# B&R Automation Studio project IP001
Automation Studio 4.7.3.93 SP

## Configuration Config1

CPU X20CP1301, AutomationRuntime C4.72, Build 4.1.2, Vc V4.72.0

### Hardware
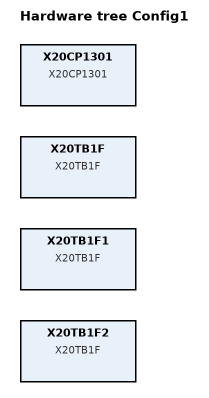
```
X20CP1301 : X20CP1301 v1.6.1.0  [X1 -> X1.SL; X2 -> X2.SL; X3 -> X3.SL]
  Module X1 (Type=X1, Virtual=true, Version=1.6.1.0)
    Connection (Connector=SS1, TargetModule=X20TB1F, TargetConnector=SS)
    Connection (Connector=SL, TargetModule=X20CP1301, TargetConnector=X1)
  Module X2 (Type=X2, Virtual=true, Version=1.6.1.0)
    Connection (Connector=SS1, TargetModule=X20TB1F1, TargetConnector=SS)
    Connection (Connector=SL, TargetModule=X20CP1301, TargetConnector=X2)
  Module X3 (Type=X3, Virtual=true, Version=1.6.1.0)
    Connection (Connector=SS1, TargetModule=X20TB1F2, TargetConnector=SS)
    Connection (Connector=SL, TargetModule=X20CP1301, TargetConnector=X3)
  Connector IF2:
    ActivateDevice = 1
    Mode = Manual
    InternetAddress = 192.168.15.199
    SubnetMask = 255.255.255.0
  ConfigurationID = IP001_Config1
  EthernetDefaultGateway = 192.168.15.254
  ActivateOpcUa = 1
  OpcUaInformationModels_PV_Version = 1
X20TB1F : X20TB1F v1.0.0.0
X20TB1F1 : X20TB1F v1.0.0.0
X20TB1F2 : X20TB1F v1.0.0.0
```

## Configuration DCS13_1

### Task classes (Cpu.sw)
```
Cyclic#4 (cycle 100000 us, tolerance 100000 us):
  DCS13_1 <- DCS13_1.prg
Libraries: Lib489, standard, AsMbTCP, operator, astime, AsIecCon, LibIP001, AsBrStr, asstring, MTBasics, DRV_mbus, DataObj, sys_lib, brsystem, MTTypes, dvframe, runtime
```

### Hardware
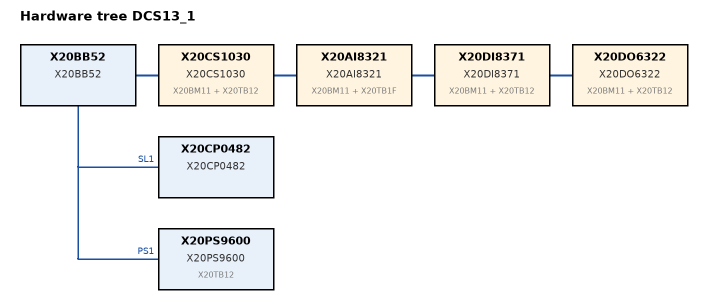
```
X20AI8321 : X20AI8321 v1.4.0.0  [SS1 -> X20TB1F.SS; SL -> X20BM11a.SL1]
X20BB52 : X20BB52 v1.1.0.0
X20BM11 : X20BM11 v1.0.0.1  [X2X1 -> X20BB52.IF6]
X20BM11a : X20BM11 v1.0.0.1  [X2X1 -> X20BM11.X2X2]
X20BM11b : X20BM11 v1.0.0.1  [X2X1 -> X20BM11a.X2X2]
X20BM11c : X20BM11 v1.0.0.1  [X2X1 -> X20BM11b.X2X2]
X20CP0482 : X20CP0482 v1.2.1.0  [SL -> X20BB52.SL1]
  Connector IF2:
    ActivateDevice = 1
    Mode = Manual
    InternetAddress = 192.168.50.15
    SubnetMask = 255.255.255.0
  ConfigurationID = IP001_DCS2_2
  TimerDeviceType = SWIOTIMER
  Cyclic1Duration = 10000
  Cyclic1Tolerance = 10000
  Cyclic2Duration = 20000
  Cyclic2Tolerance = 20000
  Cyclic3Duration = 50000
  Cyclic3Tolerance = 50000
  Cyclic4Duration = 100000
  Cyclic4Tolerance = 100000
  Cyclic5Duration = 200000
  Cyclic5Tolerance = 200000
  Cyclic6Duration = 500000
  Cyclic6Tolerance = 500000
  Cyclic7Duration = 1000000
  Cyclic7Tolerance = 1000000
  Cyclic8Duration = 10000
  Cyclic8Tolerance = 30000000
  ActivateOpcUa = 1
  OpcUa_AuthenticationSecurityPolicy_EnableNone = 1
  OpcUa_AuthenticationSecurityPolicy_EnableBasic128Rsa15 = 1
  OpcUaInformationModels_PV_Version = 1
X20CS1030 : X20CS1030 v1.7.0.0  [SS1 -> X20TB12a.SS; SL -> X20BM11.SL1]
X20DI8371 : X20DI8371 v1.0.2.0  [SS1 -> X20TB12b.SS; SL -> X20BM11b.SL1]
X20DO6322 : X20DO6322 v1.0.4.0  [SS1 -> X20TB12c.SS; SL -> X20BM11c.SL1]
X20PS9600 : X20PS9600 v1.0.2.0  [PS -> X20BB52.PS1; SS1 -> X20TB12.SS]
X20TB12 : X20TB12 v1.0.0.0
X20TB12a : X20TB12 v1.0.0.0
X20TB12b : X20TB12 v1.0.0.0
X20TB12c : X20TB12 v1.0.0.0
X20TB1F : X20TB1F v1.0.0.0
```

### IoMap.iom - X20CP0482/IoMap.iom
```iecst
VAR_CONFIG
	::DCS13_1:DI[1,1].In AT %IX."X20DI8371".DigitalInput01;
	::DCS13_1:DI[1,2].In AT %IX."X20DI8371".DigitalInput02;
	::DCS13_1:DI[1,3].In AT %IX."X20DI8371".DigitalInput03;
	::DCS13_1:DI[1,4].In AT %IX."X20DI8371".DigitalInput04;
	::DCS13_1:DO_[1,1].Out AT %QX."X20DO6322".DigitalOutput01;
	::DCS13_1:DO_[1,2].Out AT %QX."X20DO6322".DigitalOutput02;
	::DCS13_1:DO_[1,3].Out AT %QX."X20DO6322".DigitalOutput03;
	::DCS13_1:DO_[1,4].Out AT %QX."X20DO6322".DigitalOutput04;
	::DCS13_1:DO_[1,5].Out AT %QX."X20DO6322".DigitalOutput05;
	::DCS13_1:DO_[1,6].Out AT %QX."X20DO6322".DigitalOutput06;
	::DCS13_1:AI[1,1].RAW AT %IW."X20AI8321".AnalogInput01;
	::DCS13_1:AI[1,2].RAW AT %IW."X20AI8321".AnalogInput02;
	::DCS13_1:AI[1,3].RAW AT %IW."X20AI8321".AnalogInput03;
	::DCS13_1:AI[1,4].RAW AT %IW."X20AI8321".AnalogInput04;
	::DCS13_1:AI[1,5].RAW AT %IW."X20AI8321".AnalogInput05;
	::DCS13_1:AI[1,6].RAW AT %IW."X20AI8321".AnalogInput06;
	::DCS13_1:AI[1,7].RAW AT %IW."X20AI8321".AnalogInput07;
	::DCS13_1:AI[1,8].RAW AT %IW."X20AI8321".AnalogInput08;
	::DCS13_1:DI[1,5].In AT %IX."X20DI8371".DigitalInput05;
	::DCS13_1:DI[1,6].In AT %IX."X20DI8371".DigitalInput06;
	::DCS13_1:DI[1,7].In AT %IX."X20DI8371".DigitalInput07;
	::DCS13_1:DI[1,8].In AT %IX."X20DI8371".DigitalInput08;
END_VAR
```

## Configuration DCS15_1

CPU X20CP0482, AutomationRuntime C4.72, Build 4.1.2, Vc V4.72.0

### Task classes (Cpu.sw)
```
Cyclic#4 (cycle 100000 us, tolerance 100000 us):
  DCS15_1 <- DCS15_1.prg
Libraries: Lib489, standard, AsMbTCP, AsBrStr, asstring, operator, astime, AsIecCon, LibIP001, MTBasics, DRV_mbus, DataObj, sys_lib, brsystem, MTTypes, dvframe, runtime
```

### Hardware
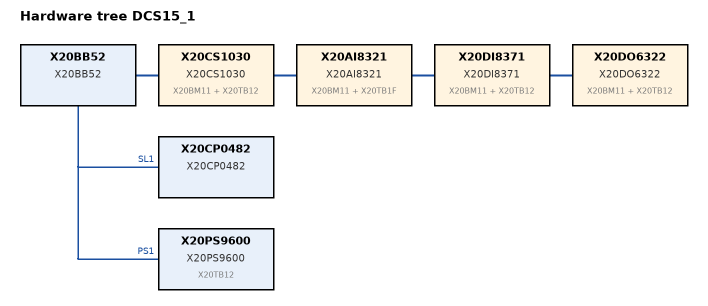
```
X20AI8321 : X20AI8321 v1.4.0.0  [SS1 -> X20TB1F.SS; SL -> X20BM11a.SL1]
X20BB52 : X20BB52 v1.1.0.0
X20BM11 : X20BM11 v1.0.0.1  [X2X1 -> X20BB52.IF6]
X20BM11a : X20BM11 v1.0.0.1  [X2X1 -> X20BM11.X2X2]
X20BM11b : X20BM11 v1.0.0.1  [X2X1 -> X20BM11a.X2X2]
X20BM11c : X20BM11 v1.0.0.1  [X2X1 -> X20BM11b.X2X2]
X20CP0482 : X20CP0482 v1.2.1.0  [SL -> X20BB52.SL1]
  Connector IF2:
    ActivateDevice = 1
    Mode = Manual
    InternetAddress = 192.168.50.16
    SubnetMask = 255.255.255.0
  ConfigurationID = IP001_DCS2_2
  TimerDeviceType = SWIOTIMER
  Cyclic1Duration = 10000
  Cyclic1Tolerance = 10000
  Cyclic2Duration = 20000
  Cyclic2Tolerance = 20000
  Cyclic3Duration = 50000
  Cyclic3Tolerance = 50000
  Cyclic4Duration = 100000
  Cyclic4Tolerance = 100000
  Cyclic5Duration = 200000
  Cyclic5Tolerance = 200000
  Cyclic6Duration = 500000
  Cyclic6Tolerance = 500000
  Cyclic7Duration = 1000000
  Cyclic7Tolerance = 1000000
  Cyclic8Duration = 10000
  Cyclic8Tolerance = 30000000
  ActivateOpcUa = 1
  OpcUa_AuthenticationSecurityPolicy_EnableNone = 1
  OpcUa_AuthenticationSecurityPolicy_EnableBasic128Rsa15 = 1
  OpcUaInformationModels_PV_Version = 1
X20CS1030 : X20CS1030 v1.7.0.0  [SS1 -> X20TB12a.SS; SL -> X20BM11.SL1]
X20DI8371 : X20DI8371 v1.0.2.0  [SS1 -> X20TB12b.SS; SL -> X20BM11b.SL1]
X20DO6322 : X20DO6322 v1.0.4.0  [SS1 -> X20TB12c.SS; SL -> X20BM11c.SL1]
X20PS9600 : X20PS9600 v1.0.2.0  [PS -> X20BB52.PS1; SS1 -> X20TB12.SS]
X20TB12 : X20TB12 v1.0.0.0
X20TB12a : X20TB12 v1.0.0.0
X20TB12b : X20TB12 v1.0.0.0
X20TB12c : X20TB12 v1.0.0.0
X20TB1F : X20TB1F v1.0.0.0
```

### IoMap.iom - X20CP0482/IoMap.iom
```iecst
VAR_CONFIG
	::DCS15_1:DI[1,1].In AT %IX."X20DI8371".DigitalInput01;
	::DCS15_1:DI[1,2].In AT %IX."X20DI8371".DigitalInput02;
	::DCS15_1:DI[1,3].In AT %IX."X20DI8371".DigitalInput03;
	::DCS15_1:DI[1,4].In AT %IX."X20DI8371".DigitalInput04;
	::DCS15_1:DO_[1,1].Out AT %QX."X20DO6322".DigitalOutput01;
	::DCS15_1:DO_[1,2].Out AT %QX."X20DO6322".DigitalOutput02;
	::DCS15_1:DO_[1,3].Out AT %QX."X20DO6322".DigitalOutput03;
	::DCS15_1:DO_[1,4].Out AT %QX."X20DO6322".DigitalOutput04;
	::DCS15_1:DO_[1,5].Out AT %QX."X20DO6322".DigitalOutput05;
	::DCS15_1:DO_[1,6].Out AT %QX."X20DO6322".DigitalOutput06;
	::DCS15_1:AI[1,1].RAW AT %IW."X20AI8321".AnalogInput01;
	::DCS15_1:AI[1,2].RAW AT %IW."X20AI8321".AnalogInput02;
	::DCS15_1:AI[1,3].RAW AT %IW."X20AI8321".AnalogInput03;
	::DCS15_1:AI[1,4].RAW AT %IW."X20AI8321".AnalogInput04;
	::DCS15_1:AI[1,5].RAW AT %IW."X20AI8321".AnalogInput05;
	::DCS15_1:AI[1,6].RAW AT %IW."X20AI8321".AnalogInput06;
	::DCS15_1:AI[1,7].RAW AT %IW."X20AI8321".AnalogInput07;
	::DCS15_1:AI[1,8].RAW AT %IW."X20AI8321".AnalogInput08;
	::DCS15_1:DI[1,5].In AT %IX."X20DI8371".DigitalInput05;
	::DCS15_1:DI[1,6].In AT %IX."X20DI8371".DigitalInput06;
	::DCS15_1:DI[1,7].In AT %IX."X20DI8371".DigitalInput07;
	::DCS15_1:DI[1,8].In AT %IX."X20DI8371".DigitalInput08;
END_VAR
```

## Configuration DCS18_1

### Hardware
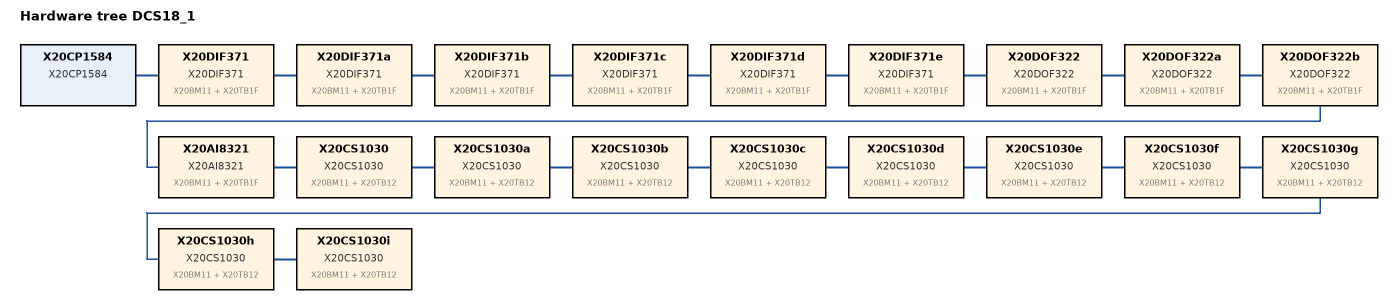
```
X20AI8321 : X20AI8321 v1.4.0.0  [SS1 -> X20TB1F.SS; SL -> X20BM11a.SL1]
X20BM11 : X20BM11 v1.0.0.1  [X2X1 -> X20BM11a.X2X2]
X20BM11a : X20BM11 v1.0.0.1  [X2X1 -> X20BM11l.X2X2]
X20BM11b : X20BM11 v1.0.0.1  [X2X1 -> X20CP1584.IF6]
X20BM11c : X20BM11 v1.0.0.1  [X2X1 -> X20BM11m.X2X2]
X20BM11d : X20BM11 v1.0.0.1  [X2X1 -> X20BM11g.X2X2]
X20BM11e : X20BM11 v1.0.0.1  [X2X1 -> X20BM11d.X2X2]
X20BM11f : X20BM11 v1.0.0.1  [X2X1 -> X20BM11c.X2X2]
X20BM11g : X20BM11 v1.0.0.1  [X2X1 -> X20BM11.X2X2]
X20BM11h : X20BM11 v1.0.0.1  [X2X1 -> X20BM11b.X2X2]
X20BM11i : X20BM11 v1.0.0.1  [X2X1 -> X20BM11h.X2X2]
X20BM11j : X20BM11 v1.0.0.1  [X2X1 -> X20BM11i.X2X2]
X20BM11k : X20BM11 v1.0.0.1  [X2X1 -> X20BM11j.X2X2]
X20BM11l : X20BM11 v1.0.0.1  [X2X1 -> X20BM11f.X2X2]
X20BM11m : X20BM11 v1.0.0.1  [X2X1 -> X20BM11k.X2X2]
X20BM11n : X20BM11 v1.0.0.1  [X2X1 -> X20BM11e.X2X2]
X20BM11o : X20BM11 v1.0.0.1  [X2X1 -> X20BM11n.X2X2]
X20BM11p : X20BM11 v1.0.0.1  [X2X1 -> X20BM11o.X2X2]
X20BM11q : X20BM11 v1.0.0.1  [X2X1 -> X20BM11p.X2X2]
X20BM11r : X20BM11 v1.0.0.1  [X2X1 -> X20BM11q.X2X2]
X20BM11s : X20BM11 v1.0.0.1  [X2X1 -> X20BM11r.X2X2]
X20CP1584 : X20CP1584 v1.8.0.0
  Connector IF2:
    ActivateDevice = 1
    Mode = Manual
    InternetAddress = 192.168.50.17
    SubnetMask = 255.255.255.0
  ConfigurationID = IP001_DCS2_2
  ActivateOpcUa = 1
  OpcUa_AuthenticationSecurityPolicy_EnableNone = 1
  OpcUa_AuthenticationSecurityPolicy_EnableBasic128Rsa15 = 1
  OpcUaInformationModels_PV_Version = 1
X20CS1030 : X20CS1030 v1.7.0.0  [SS1 -> X20TB12a.SS; SL -> X20BM11.SL1]
X20CS1030a : X20CS1030 v1.7.0.0  [SS1 -> X20TB12.SS; SL -> X20BM11g.SL1]
X20CS1030b : X20CS1030 v1.7.0.0  [SS1 -> X20TB12b.SS; SL -> X20BM11d.SL1]
X20CS1030c : X20CS1030 v1.7.0.0  [SS1 -> X20TB12c.SS; SL -> X20BM11e.SL1]
X20CS1030d : X20CS1030 v1.7.0.0  [SS1 -> X20TB12d.SS; SL -> X20BM11n.SL1]
X20CS1030e : X20CS1030 v1.7.0.0  [SS1 -> X20TB12e.SS; SL -> X20BM11o.SL1]
X20CS1030f : X20CS1030 v1.7.0.0  [SS1 -> X20TB12f.SS; SL -> X20BM11p.SL1]
X20CS1030g : X20CS1030 v1.7.0.0  [SS1 -> X20TB12g.SS; SL -> X20BM11q.SL1]
X20CS1030h : X20CS1030 v1.7.0.0  [SS1 -> X20TB12h.SS; SL -> X20BM11r.SL1]
X20CS1030i : X20CS1030 v1.7.0.0  [SS1 -> X20TB12i.SS; SL -> X20BM11s.SL1]
X20DIF371 : X20DIF371 v1.1.0.0  [SS1 -> X20TB1F1.SS; SL -> X20BM11b.SL1]
X20DIF371a : X20DIF371 v1.1.0.0  [SS1 -> X20TB1F2.SS; SL -> X20BM11h.SL1]
X20DIF371b : X20DIF371 v1.1.0.0  [SS1 -> X20TB1F3.SS; SL -> X20BM11i.SL1]
X20DIF371c : X20DIF371 v1.1.0.0  [SS1 -> X20TB1F4.SS; SL -> X20BM11j.SL1]
X20DIF371d : X20DIF371 v1.1.0.0  [SS1 -> X20TB1F5.SS; SL -> X20BM11k.SL1]
X20DIF371e : X20DIF371 v1.1.0.0  [SS1 -> X20TB1F9.SS; SL -> X20BM11m.SL1]
X20DOF322 : X20DOF322 v1.4.0.0  [SS1 -> X20TB1F6.SS; SL -> X20BM11c.SL1]
X20DOF322a : X20DOF322 v1.4.0.0  [SS1 -> X20TB1F7.SS; SL -> X20BM11f.SL1]
X20DOF322b : X20DOF322 v1.4.0.0  [SS1 -> X20TB1F8.SS; SL -> X20BM11l.SL1]
X20TB12 : X20TB12 v1.0.0.0
X20TB12a : X20TB12 v1.0.0.0
X20TB12b : X20TB12 v1.0.0.0
X20TB12c : X20TB12 v1.0.0.0
X20TB12d : X20TB12 v1.0.0.0
X20TB12e : X20TB12 v1.0.0.0
X20TB12f : X20TB12 v1.0.0.0
X20TB12g : X20TB12 v1.0.0.0
X20TB12h : X20TB12 v1.0.0.0
X20TB12i : X20TB12 v1.0.0.0
X20TB1F : X20TB1F v1.0.0.0
X20TB1F1 : X20TB1F v1.0.0.0
X20TB1F2 : X20TB1F v1.0.0.0
X20TB1F3 : X20TB1F v1.0.0.0
X20TB1F4 : X20TB1F v1.0.0.0
X20TB1F5 : X20TB1F v1.0.0.0
X20TB1F6 : X20TB1F v1.0.0.0
X20TB1F7 : X20TB1F v1.0.0.0
X20TB1F8 : X20TB1F v1.0.0.0
X20TB1F9 : X20TB1F v1.0.0.0
```

### IoMap.iom - X20CP1584/IoMap.iom
```iecst
VAR_CONFIG
	::DCS18_1:AI[1,1].RAW AT %IW."X20AI8321".AnalogInput01;
	::DCS18_1:AI[1,2].RAW AT %IW."X20AI8321".AnalogInput02;
	::DCS18_1:AI[1,3].RAW AT %IW."X20AI8321".AnalogInput03;
	::DCS18_1:AI[1,4].RAW AT %IW."X20AI8321".AnalogInput04;
	::DCS18_1:AI[1,5].RAW AT %IW."X20AI8321".AnalogInput05;
	::DCS18_1:AI[1,6].RAW AT %IW."X20AI8321".AnalogInput06;
	::DCS18_1:AI[1,7].RAW AT %IW."X20AI8321".AnalogInput07;
	::DCS18_1:AI[1,8].RAW AT %IW."X20AI8321".AnalogInput08;
	::DCS18_1:DI[1,1].In AT %IX."X20DIF371".DigitalInput01;
	::DCS18_1:DI[1,2].In AT %IX."X20DIF371".DigitalInput02;
	::DCS18_1:DI[1,3].In AT %IX."X20DIF371".DigitalInput03;
	::DCS18_1:DI[1,4].In AT %IX."X20DIF371".DigitalInput04;
	::DCS18_1:DI[1,5].In AT %IX."X20DIF371".DigitalInput05;
	::DCS18_1:DI[1,6].In AT %IX."X20DIF371".DigitalInput06;
	::DCS18_1:DI[1,7].In AT %IX."X20DIF371".DigitalInput07;
	::DCS18_1:DI[1,8].In AT %IX."X20DIF371".DigitalInput08;
	::DCS18_1:DI[1,9].In AT %IX."X20DIF371".DigitalInput09;
	::DCS18_1:DI[1,10].In AT %IX."X20DIF371".DigitalInput10;
	::DCS18_1:DI[1,11].In AT %IX."X20DIF371".DigitalInput11;
	::DCS18_1:DI[1,12].In AT %IX."X20DIF371".DigitalInput12;
	::DCS18_1:DI[1,13].In AT %IX."X20DIF371".DigitalInput13;
	::DCS18_1:DI[1,14].In AT %IX."X20DIF371".DigitalInput14;
	::DCS18_1:DI[1,15].In AT %IX."X20DIF371".DigitalInput15;
	::DCS18_1:DI[1,16].In AT %IX."X20DIF371".DigitalInput16;
	::DCS18_1:DO_[1,1].Out AT %QX."X20DOF322".DigitalOutput01;
	::DCS18_1:DO_[1,2].Out AT %QX."X20DOF322".DigitalOutput02;
	::DCS18_1:DO_[1,3].Out AT %QX."X20DOF322".DigitalOutput03;
	::DCS18_1:DO_[1,4].Out AT %QX."X20DOF322".DigitalOutput04;
	::DCS18_1:DO_[1,5].Out AT %QX."X20DOF322".DigitalOutput05;
	::DCS18_1:DO_[1,6].Out AT %QX."X20DOF322".DigitalOutput06;
	::DCS18_1:DO_[1,7].Out AT %QX."X20DOF322".DigitalOutput07;
	::DCS18_1:DO_[1,8].Out AT %QX."X20DOF322".DigitalOutput08;
	::DCS18_1:DO_[1,9].Out AT %QX."X20DOF322".DigitalOutput09;
	::DCS18_1:DO_[1,10].Out AT %QX."X20DOF322".DigitalOutput10;
	::DCS18_1:DO_[1,11].Out AT %QX."X20DOF322".DigitalOutput11;
	::DCS18_1:DO_[1,12].Out AT %QX."X20DOF322".DigitalOutput12;
	::DCS18_1:DO_[1,13].Out AT %QX."X20DOF322".DigitalOutput13;
	::DCS18_1:DO_[1,14].Out AT %QX."X20DOF322".DigitalOutput14;
	::DCS18_1:DO_[1,15].Out AT %QX."X20DOF322".DigitalOutput15;
	::DCS18_1:DO_[1,16].Out AT %QX."X20DOF322".DigitalOutput16;
	::DCS18_1:DO_[2,1].Out AT %QX."X20DOF322a".DigitalOutput01;
	::DCS18_1:DO_[2,2].Out AT %QX."X20DOF322a".DigitalOutput02;
	::DCS18_1:DO_[2,3].Out AT %QX."X20DOF322a".DigitalOutput03;
	::DCS18_1:DO_[2,4].Out  AT %QX."X20DOF322a".DigitalOutput04;
	::DCS18_1:DO_[2,5].Out  AT %QX."X20DOF322a".DigitalOutput05;
	::DCS18_1:DO_[2,6].Out  AT %QX."X20DOF322a".DigitalOutput06;
	::DCS18_1:DO_[2,7].Out  AT %QX."X20DOF322a".DigitalOutput07;
	::DCS18_1:DO_[2,8].Out  AT %QX."X20DOF322a".DigitalOutput08;
	::DCS18_1:DO_[2,9].Out  AT %QX."X20DOF322a".DigitalOutput09;
	::DCS18_1:DO_[2,10].Out  AT %QX."X20DOF322a".DigitalOutput10;
	::DCS18_1:DO_[2,11].Out  AT %QX."X20DOF322a".DigitalOutput11;
	::DCS18_1:DO_[2,12].Out  AT %QX."X20DOF322a".DigitalOutput12;
	::DCS18_1:DO_[2,13].Out  AT %QX."X20DOF322a".DigitalOutput13;
	::DCS18_1:DO_[2,14].Out  AT %QX."X20DOF322a".DigitalOutput14;
	::DCS18_1:DO_[2,15].Out  AT %QX."X20DOF322a".DigitalOutput15;
	::DCS18_1:DO_[2,16].Out  AT %QX."X20DOF322a".DigitalOutput16;
	::DCS18_1:DO_[3,1].Out AT %QX."X20DOF322b".DigitalOutput01;
	::DCS18_1:DO_[3,2].Out  AT %QX."X20DOF322b".DigitalOutput02;
	::DCS18_1:DO_[3,3].Out  AT %QX."X20DOF322b".DigitalOutput03;
	::DCS18_1:DO_[3,4].Out  AT %QX."X20DOF322b".DigitalOutput04;
	::DCS18_1:DO_[3,5].Out  AT %QX."X20DOF322b".DigitalOutput05;
	::DCS18_1:DO_[3,6].Out  AT %QX."X20DOF322b".DigitalOutput06;
	::DCS18_1:DO_[3,7].Out  AT %QX."X20DOF322b".DigitalOutput07;
	::DCS18_1:DO_[3,8].Out  AT %QX."X20DOF322b".DigitalOutput08;
	::DCS18_1:DO_[3,9].Out  AT %QX."X20DOF322b".DigitalOutput09;
	::DCS18_1:DO_[3,10].Out  AT %QX."X20DOF322b".DigitalOutput10;
	::DCS18_1:DO_[3,11].Out  AT %QX."X20DOF322b".DigitalOutput11;
	::DCS18_1:DO_[3,12].Out  AT %QX."X20DOF322b".DigitalOutput12;
	::DCS18_1:DO_[3,13].Out  AT %QX."X20DOF322b".DigitalOutput13;
	::DCS18_1:DO_[3,14].Out  AT %QX."X20DOF322b".DigitalOutput14;
	::DCS18_1:DO_[3,15].Out  AT %QX."X20DOF322b".DigitalOutput15;
	::DCS18_1:DO_[3,16].Out  AT %QX."X20DOF322b".DigitalOutput16;
END_VAR
```

## Configuration DCS2_2

CPU X20CP0482, AutomationRuntime B4.92, Build 4.1.2, Vc V4.72.5

### Task classes (Cpu.sw)
```
Cyclic#4 (cycle 100000 us, tolerance 100000 us):
  DCS2_2 <- DCS2_2.prg
Libraries: Lib489, standard, AsMbTCP, AsBrStr, asstring, MTBasics, DRV_mbus, DataObj, sys_lib, brsystem, MTTypes, dvframe, runtime, LibIP001
```

### Hardware
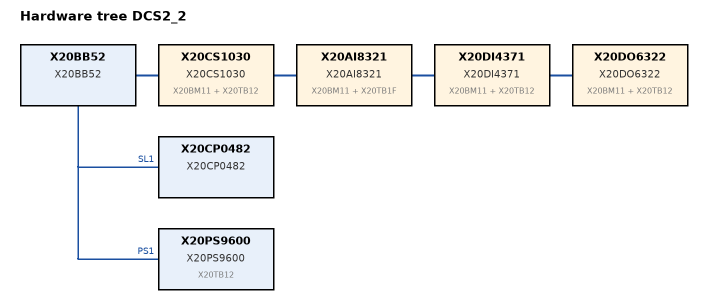
```
X20AI8321 : X20AI8321 v1.5.0.0  [SS1 -> X20TB1F.SS; SL -> X20BM11a.SL1]
X20BB52 : X20BB52 v1.2.0.0
X20BM11 : X20BM11 v1.1.0.0  [X2X1 -> X20BB52.IF6]
X20BM11a : X20BM11 v1.1.0.0  [X2X1 -> X20BM11.X2X2]
X20BM11b : X20BM11 v1.1.0.0  [X2X1 -> X20BM11a.X2X2]
X20BM11c : X20BM11 v1.1.0.0  [X2X1 -> X20BM11b.X2X2]
X20CP0482 : X20CP0482 v1.5.0.0  [SL -> X20BB52.SL1]
  Connector IF2:
    ActivateDevice = 1
    Mode = Manual
    InternetAddress = 192.168.50.10
    SubnetMask = 255.255.255.0
  Connector IF3:
    DNAConfiguration = manual
  ConfigurationID = IP001_DCS2_2
  UserPartitionSize = 0
  Simulation = 1
  TimerDeviceType = SWIOTIMER
  Cyclic1Duration = 10000
  Cyclic1Tolerance = 10000
  Cyclic2Duration = 20000
  Cyclic2Tolerance = 20000
  Cyclic3Duration = 50000
  Cyclic3Tolerance = 50000
  Cyclic4Duration = 100000
  Cyclic4Tolerance = 100000
  Cyclic5Duration = 200000
  Cyclic5Tolerance = 200000
  Cyclic6Duration = 500000
  Cyclic6Tolerance = 500000
  Cyclic7Duration = 1000000
  Cyclic7Tolerance = 1000000
  Cyclic8Duration = 10000
  Cyclic8Tolerance = 30000000
  FileDevice1
  FileDeviceName1 = USER
  FileDevicePath1 = USER_PATH
  ActivateOpcUa = 1
  OpcUa_AuthenticationSecurityPolicy_EnableNone = 1
  OpcUa_AuthenticationSecurityPolicy_EnableBasic128Rsa15 = 1
  OpcUaInformationModels_PV_Version = 1
X20CS1030 : X20CS1030 v1.8.0.0  [SS1 -> X20TB12a.SS; SL -> X20BM11.SL1]
X20DI4371 : X20DI4371 v1.2.0.0  [SS1 -> X20TB12b.SS; SL -> X20BM11b.SL1]
X20DO6322 : X20DO6322 v1.2.0.0  [SS1 -> X20TB12c.SS; SL -> X20BM11c.SL1]
X20PS9600 : X20PS9600 v1.6.0.0  [PS -> X20BB52.PS1; SS1 -> X20TB12.SS]
X20TB12 : X20TB12 v1.0.0.0
X20TB12a : X20TB12 v1.0.0.0
X20TB12b : X20TB12 v1.0.0.0
X20TB12c : X20TB12 v1.0.0.0
X20TB1F : X20TB1F v1.0.0.0
```

### IoMap.iom - X20CP0482/IoMap.iom
```iecst
VAR_CONFIG
	::DCS2_2:AI[1,1].RAW AT %IW."X20AI8321".AnalogInput01;
	::DCS2_2:AI[1,2].RAW  AT %IW."X20AI8321".AnalogInput02;
	::DCS2_2:AI[1,3].RAW AT %IW."X20AI8321".AnalogInput03;
	::DCS2_2:AI[1,4].RAW AT %IW."X20AI8321".AnalogInput04;
	::DCS2_2:AI[1,5].RAW AT %IW."X20AI8321".AnalogInput05;
	::DCS2_2:AI[1,6].RAW AT %IW."X20AI8321".AnalogInput06;
	::DCS2_2:AI[1,7].RAW AT %IW."X20AI8321".AnalogInput07;
	::DCS2_2:AI[1,8].RAW AT %IW."X20AI8321".AnalogInput08;
	::DCS2_2:DI[1,1].In AT %IX."X20DI4371".DigitalInput01;
	::DCS2_2:DI[1,2].In AT %IX."X20DI4371".DigitalInput02;
	::DCS2_2:DI[1,3].In AT %IX."X20DI4371".DigitalInput03;
	::DCS2_2:DI[1,4].In AT %IX."X20DI4371".DigitalInput04;
	::DCS2_2:DO_[1,1].Out AT %QX."X20DO6322".DigitalOutput01;
	::DCS2_2:DO_[1,2].Out AT %QX."X20DO6322".DigitalOutput02;
	::DCS2_2:DO_[1,3].Out AT %QX."X20DO6322".DigitalOutput03;
	::DCS2_2:DO_[1,4].Out AT %QX."X20DO6322".DigitalOutput04;
	::DCS2_2:DO_[1,5].Out AT %QX."X20DO6322".DigitalOutput05;
	::DCS2_2:DO_[1,6].Out AT %QX."X20DO6322".DigitalOutput06;
END_VAR
```

## Configuration DCS31_1

CPU X20CP0482, AutomationRuntime C4.72, Build 4.1.2, Vc V4.72.0

### Task classes (Cpu.sw)
```
Cyclic#4 (cycle 100000 us, tolerance 100000 us):
  DCS31_1 <- DCS31_1.prg
Libraries: Lib489, standard, AsMbTCP, AsBrStr, asstring, operator, astime, AsIecCon, LibIP001, MTBasics, DRV_mbus, DataObj, sys_lib, brsystem, MTTypes, dvframe, runtime
```

### Hardware
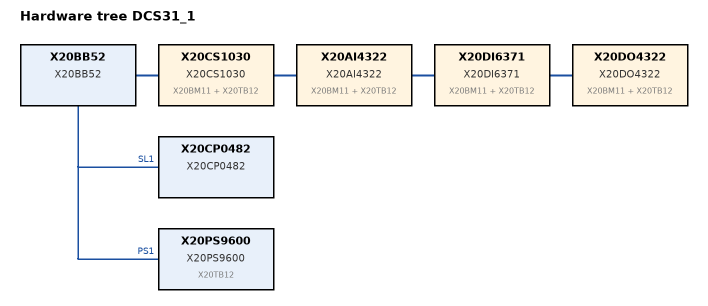
```
X20AI4322 : X20AI4322 v1.0.0.2  [SS1 -> X20TB12d.SS; SL -> X20BM11a.SL1]
X20BB52 : X20BB52 v1.1.0.0
X20BM11 : X20BM11 v1.0.0.1  [X2X1 -> X20BB52.IF6]
X20BM11a : X20BM11 v1.0.0.1  [X2X1 -> X20BM11.X2X2]
X20BM11b : X20BM11 v1.0.0.1  [X2X1 -> X20BM11a.X2X2]
X20BM11c : X20BM11 v1.0.0.1  [X2X1 -> X20BM11b.X2X2]
X20CP0482 : X20CP0482 v1.2.1.0  [SL -> X20BB52.SL1]
  Connector IF2:
    ActivateDevice = 1
    Mode = Manual
    InternetAddress = 192.168.50.18
    SubnetMask = 255.255.255.0
  ConfigurationID = IP001_DCS2_2
  TimerDeviceType = SWIOTIMER
  Cyclic1Duration = 10000
  Cyclic1Tolerance = 10000
  Cyclic2Duration = 20000
  Cyclic2Tolerance = 20000
  Cyclic3Duration = 50000
  Cyclic3Tolerance = 50000
  Cyclic4Duration = 100000
  Cyclic4Tolerance = 100000
  Cyclic5Duration = 200000
  Cyclic5Tolerance = 200000
  Cyclic6Duration = 500000
  Cyclic6Tolerance = 500000
  Cyclic7Duration = 1000000
  Cyclic7Tolerance = 1000000
  Cyclic8Duration = 10000
  Cyclic8Tolerance = 30000000
  ActivateOpcUa = 1
  OpcUa_AuthenticationSecurityPolicy_EnableNone = 1
  OpcUa_AuthenticationSecurityPolicy_EnableBasic128Rsa15 = 1
  OpcUaInformationModels_PV_Version = 1
X20CS1030 : X20CS1030 v1.7.0.0  [SS1 -> X20TB12a.SS; SL -> X20BM11.SL1]
X20DI6371 : X20DI6371 v1.0.2.0  [SS1 -> X20TB12b.SS; SL -> X20BM11b.SL1]
X20DO4322 : X20DO4322 v1.0.3.0  [SS1 -> X20TB12c.SS; SL -> X20BM11c.SL1]
X20PS9600 : X20PS9600 v1.0.2.0  [PS -> X20BB52.PS1; SS1 -> X20TB12.SS]
X20TB12 : X20TB12 v1.0.0.0
X20TB12a : X20TB12 v1.0.0.0
X20TB12b : X20TB12 v1.0.0.0
X20TB12c : X20TB12 v1.0.0.0
X20TB12d : X20TB12 v1.0.0.0
```

### IoMap.iom - X20CP0482/IoMap.iom
```iecst
VAR_CONFIG
	::DCS31_1:DI[1,1].In AT %IX."X20DI6371".DigitalInput01;
	::DCS31_1:DI[1,2].In AT %IX."X20DI6371".DigitalInput02;
	::DCS31_1:DI[1,3].In AT %IX."X20DI6371".DigitalInput03;
	::DCS31_1:DI[1,4].In AT %IX."X20DI6371".DigitalInput04;
	::DCS31_1:DO_[1,1].Out AT %QX."X20DO4322".DigitalOutput01;
	::DCS31_1:DO_[1,2].Out AT %QX."X20DO4322".DigitalOutput02;
	::DCS31_1:DO_[1,3].Out AT %QX."X20DO4322".DigitalOutput03;
	::DCS31_1:DO_[1,4].Out AT %QX."X20DO4322".DigitalOutput04;
	::DCS31_1:AI[1,1].RAW AT %IW."X20AI4322".AnalogInput01;
	::DCS31_1:AI[1,2].RAW AT %IW."X20AI4322".AnalogInput02;
	::DCS31_1:AI[1,3].RAW AT %IW."X20AI4322".AnalogInput03;
	::DCS31_1:AI[1,4].RAW AT %IW."X20AI4322".AnalogInput04;
	::DCS31_1:DI[1,5].In AT %IX."X20DI6371".DigitalInput05;
	::DCS31_1:DI[1,6].In AT %IX."X20DI6371".DigitalInput06;
END_VAR
```

## Configuration DCS31_2

### Hardware
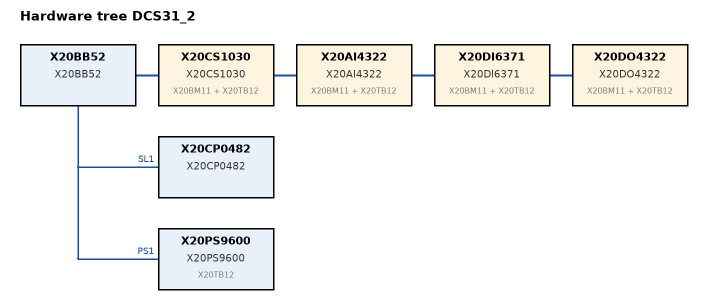
```
X20AI4322 : X20AI4322 v1.0.0.2  [SS1 -> X20TB12d.SS; SL -> X20BM11a.SL1]
X20BB52 : X20BB52 v1.1.0.0
X20BM11 : X20BM11 v1.0.0.1  [X2X1 -> X20BB52.IF6]
X20BM11a : X20BM11 v1.0.0.1  [X2X1 -> X20BM11.X2X2]
X20BM11b : X20BM11 v1.0.0.1  [X2X1 -> X20BM11a.X2X2]
X20BM11c : X20BM11 v1.0.0.1  [X2X1 -> X20BM11b.X2X2]
X20CP0482 : X20CP0482 v1.2.1.0  [SL -> X20BB52.SL1]
  Connector IF2:
    ActivateDevice = 1
    Mode = Manual
    InternetAddress = 192.168.50.19
    SubnetMask = 255.255.255.0
  ConfigurationID = IP001_DCS2_2
  TimerDeviceType = SWIOTIMER
  Cyclic1Duration = 10000
  Cyclic1Tolerance = 10000
  Cyclic2Duration = 20000
  Cyclic2Tolerance = 20000
  Cyclic3Duration = 50000
  Cyclic3Tolerance = 50000
  Cyclic4Duration = 100000
  Cyclic4Tolerance = 100000
  Cyclic5Duration = 200000
  Cyclic5Tolerance = 200000
  Cyclic6Duration = 500000
  Cyclic6Tolerance = 500000
  Cyclic7Duration = 1000000
  Cyclic7Tolerance = 1000000
  Cyclic8Duration = 10000
  Cyclic8Tolerance = 30000000
  ActivateOpcUa = 1
  OpcUa_AuthenticationSecurityPolicy_EnableNone = 1
  OpcUa_AuthenticationSecurityPolicy_EnableBasic128Rsa15 = 1
  OpcUaInformationModels_PV_Version = 1
X20CS1030 : X20CS1030 v1.7.0.0  [SS1 -> X20TB12a.SS; SL -> X20BM11.SL1]
X20DI6371 : X20DI6371 v1.0.2.0  [SS1 -> X20TB12b.SS; SL -> X20BM11b.SL1]
X20DO4322 : X20DO4322 v1.0.3.0  [SS1 -> X20TB12c.SS; SL -> X20BM11c.SL1]
X20PS9600 : X20PS9600 v1.0.2.0  [PS -> X20BB52.PS1; SS1 -> X20TB12.SS]
X20TB12 : X20TB12 v1.0.0.0
X20TB12a : X20TB12 v1.0.0.0
X20TB12b : X20TB12 v1.0.0.0
X20TB12c : X20TB12 v1.0.0.0
X20TB12d : X20TB12 v1.0.0.0
```

### IoMap.iom - X20CP0482/IoMap.iom
```iecst
VAR_CONFIG
	::DCS31_2:DI[1,1].In AT %IX."X20DI6371".DigitalInput01;
	::DCS31_2:DI[1,2].In AT %IX."X20DI6371".DigitalInput02;
	::DCS31_2:DI[1,3].In AT %IX."X20DI6371".DigitalInput03;
	::DCS31_2:DI[1,4].In AT %IX."X20DI6371".DigitalInput04;
	::DCS31_2:DO_[1,1].Out AT %QX."X20DO4322".DigitalOutput01;
	::DCS31_2:DO_[1,2].Out AT %QX."X20DO4322".DigitalOutput02;
	::DCS31_2:DO_[1,3].Out AT %QX."X20DO4322".DigitalOutput03;
	::DCS31_2:DO_[1,4].Out AT %QX."X20DO4322".DigitalOutput04;
	::DCS31_2:AI[1,1].RAW AT %IW."X20AI4322".AnalogInput01;
	::DCS31_2:AI[1,2].RAW AT %IW."X20AI4322".AnalogInput02;
	::DCS31_2:AI[1,3].RAW AT %IW."X20AI4322".AnalogInput03;
	::DCS31_2:AI[1,4].RAW AT %IW."X20AI4322".AnalogInput04;
	::DCS31_2:DI[1,5].In AT %IX."X20DI6371".DigitalInput05;
	::DCS31_2:DI[1,6].In AT %IX."X20DI6371".DigitalInput06;
END_VAR
```

## Configuration DCS31_3

### Task classes (Cpu.sw)
```
Cyclic#4 (cycle 100000 us, tolerance 100000 us):
  DCS31_3 <- DCS31_3.prg
Libraries: Lib489, standard, AsMbTCP, AsBrStr, operator, astime, AsIecCon, LibIP001, asstring, MTBasics, DRV_mbus, DataObj, sys_lib, brsystem, MTTypes, dvframe, runtime
```

### Hardware
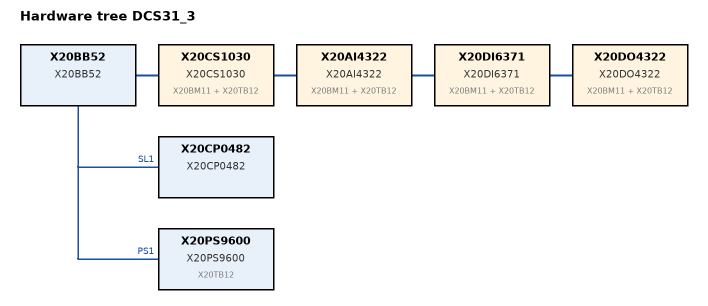
```
X20AI4322 : X20AI4322 v1.0.0.2  [SS1 -> X20TB12d.SS; SL -> X20BM11a.SL1]
X20BB52 : X20BB52 v1.1.0.0
X20BM11 : X20BM11 v1.0.0.1  [X2X1 -> X20BB52.IF6]
X20BM11a : X20BM11 v1.0.0.1  [X2X1 -> X20BM11.X2X2]
X20BM11b : X20BM11 v1.0.0.1  [X2X1 -> X20BM11a.X2X2]
X20BM11c : X20BM11 v1.0.0.1  [X2X1 -> X20BM11b.X2X2]
X20CP0482 : X20CP0482 v1.2.1.0  [SL -> X20BB52.SL1]
  Connector IF2:
    ActivateDevice = 1
    Mode = Manual
    InternetAddress = 192.168.50.20
    SubnetMask = 255.255.255.0
  ConfigurationID = IP001_DCS2_2
  TimerDeviceType = SWIOTIMER
  Cyclic1Duration = 10000
  Cyclic1Tolerance = 10000
  Cyclic2Duration = 20000
  Cyclic2Tolerance = 20000
  Cyclic3Duration = 50000
  Cyclic3Tolerance = 50000
  Cyclic4Duration = 100000
  Cyclic4Tolerance = 100000
  Cyclic5Duration = 200000
  Cyclic5Tolerance = 200000
  Cyclic6Duration = 500000
  Cyclic6Tolerance = 500000
  Cyclic7Duration = 1000000
  Cyclic7Tolerance = 1000000
  Cyclic8Duration = 10000
  Cyclic8Tolerance = 30000000
  ActivateOpcUa = 1
  OpcUa_AuthenticationSecurityPolicy_EnableNone = 1
  OpcUa_AuthenticationSecurityPolicy_EnableBasic128Rsa15 = 1
  OpcUaInformationModels_PV_Version = 1
X20CS1030 : X20CS1030 v1.7.0.0  [SS1 -> X20TB12a.SS; SL -> X20BM11.SL1]
X20DI6371 : X20DI6371 v1.0.2.0  [SS1 -> X20TB12b.SS; SL -> X20BM11b.SL1]
X20DO4322 : X20DO4322 v1.0.3.0  [SS1 -> X20TB12c.SS; SL -> X20BM11c.SL1]
X20PS9600 : X20PS9600 v1.0.2.0  [PS -> X20BB52.PS1; SS1 -> X20TB12.SS]
X20TB12 : X20TB12 v1.0.0.0
X20TB12a : X20TB12 v1.0.0.0
X20TB12b : X20TB12 v1.0.0.0
X20TB12c : X20TB12 v1.0.0.0
X20TB12d : X20TB12 v1.0.0.0
```

### IoMap.iom - X20CP0482/IoMap.iom
```iecst
VAR_CONFIG
	::DCS31_3:DI[1,1].In AT %IX."X20DI6371".DigitalInput01;
	::DCS31_3:DI[1,2].In AT %IX."X20DI6371".DigitalInput02;
	::DCS31_3:DI[1,3].In AT %IX."X20DI6371".DigitalInput03;
	::DCS31_3:DI[1,4].In AT %IX."X20DI6371".DigitalInput04;
	::DCS31_3:DO_[1,1].Out AT %QX."X20DO4322".DigitalOutput01;
	::DCS31_3:DO_[1,2].Out AT %QX."X20DO4322".DigitalOutput02;
	::DCS31_3:DO_[1,3].Out AT %QX."X20DO4322".DigitalOutput03;
	::DCS31_3:DO_[1,4].Out AT %QX."X20DO4322".DigitalOutput04;
	::DCS31_3:AI[1,1].RAW AT %IW."X20AI4322".AnalogInput01;
	::DCS31_3:AI[1,2].RAW AT %IW."X20AI4322".AnalogInput02;
	::DCS31_3:AI[1,3].RAW AT %IW."X20AI4322".AnalogInput03;
	::DCS31_3:AI[1,4].RAW AT %IW."X20AI4322".AnalogInput04;
	::DCS31_3:DI[1,5].In AT %IX."X20DI6371".DigitalInput05;
	::DCS31_3:DI[1,6].In AT %IX."X20DI6371".DigitalInput06;
END_VAR
```

## Configuration DCS31_4

CPU X20CP0482, AutomationRuntime C4.72, Build 4.1.2, Vc V4.72.0

### Hardware
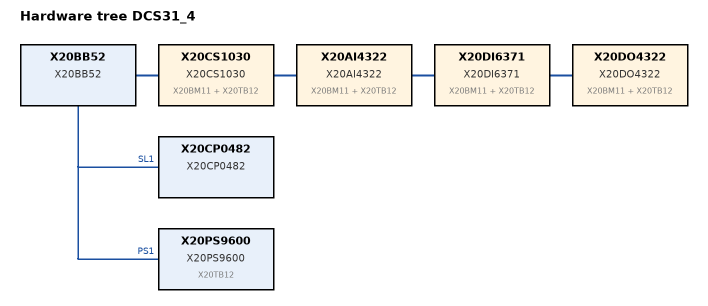
```
X20AI4322 : X20AI4322 v1.0.0.2  [SS1 -> X20TB12d.SS; SL -> X20BM11a.SL1]
X20BB52 : X20BB52 v1.1.0.0
X20BM11 : X20BM11 v1.0.0.1  [X2X1 -> X20BB52.IF6]
X20BM11a : X20BM11 v1.0.0.1  [X2X1 -> X20BM11.X2X2]
X20BM11b : X20BM11 v1.0.0.1  [X2X1 -> X20BM11a.X2X2]
X20BM11c : X20BM11 v1.0.0.1  [X2X1 -> X20BM11b.X2X2]
X20CP0482 : X20CP0482 v1.2.1.0  [SL -> X20BB52.SL1]
  Connector IF2:
    ActivateDevice = 1
    Mode = Manual
    InternetAddress = 192.168.50.21
    SubnetMask = 255.255.255.0
  ConfigurationID = IP001_DCS2_2
  TimerDeviceType = SWIOTIMER
  Cyclic1Duration = 10000
  Cyclic1Tolerance = 10000
  Cyclic2Duration = 20000
  Cyclic2Tolerance = 20000
  Cyclic3Duration = 50000
  Cyclic3Tolerance = 50000
  Cyclic4Duration = 100000
  Cyclic4Tolerance = 100000
  Cyclic5Duration = 200000
  Cyclic5Tolerance = 200000
  Cyclic6Duration = 500000
  Cyclic6Tolerance = 500000
  Cyclic7Duration = 1000000
  Cyclic7Tolerance = 1000000
  Cyclic8Duration = 10000
  Cyclic8Tolerance = 30000000
  ActivateOpcUa = 1
  OpcUa_AuthenticationSecurityPolicy_EnableNone = 1
  OpcUa_AuthenticationSecurityPolicy_EnableBasic128Rsa15 = 1
  OpcUaInformationModels_PV_Version = 1
X20CS1030 : X20CS1030 v1.7.0.0  [SS1 -> X20TB12a.SS; SL -> X20BM11.SL1]
X20DI6371 : X20DI6371 v1.0.2.0  [SS1 -> X20TB12b.SS; SL -> X20BM11b.SL1]
X20DO4322 : X20DO4322 v1.0.3.0  [SS1 -> X20TB12c.SS; SL -> X20BM11c.SL1]
X20PS9600 : X20PS9600 v1.0.2.0  [PS -> X20BB52.PS1; SS1 -> X20TB12.SS]
X20TB12 : X20TB12 v1.0.0.0
X20TB12a : X20TB12 v1.0.0.0
X20TB12b : X20TB12 v1.0.0.0
X20TB12c : X20TB12 v1.0.0.0
X20TB12d : X20TB12 v1.0.0.0
```

### IoMap.iom - X20CP0482/IoMap.iom
```iecst
VAR_CONFIG
	::DCS31_4:DI[1,1].In AT %IX."X20DI6371".DigitalInput01;
	::DCS31_4:DI[1,2].In AT %IX."X20DI6371".DigitalInput02;
	::DCS31_4:DI[1,3].In AT %IX."X20DI6371".DigitalInput03;
	::DCS31_4:DI[1,4].In AT %IX."X20DI6371".DigitalInput04;
	::DCS31_4:DO_[1,1].Out AT %QX."X20DO4322".DigitalOutput01;
	::DCS31_4:DO_[1,2].Out AT %QX."X20DO4322".DigitalOutput02;
	::DCS31_4:DO_[1,3].Out AT %QX."X20DO4322".DigitalOutput03;
	::DCS31_4:DO_[1,4].Out AT %QX."X20DO4322".DigitalOutput04;
	::DCS31_4:AI[1,1].RAW AT %IW."X20AI4322".AnalogInput01;
	::DCS31_4:AI[1,2].RAW AT %IW."X20AI4322".AnalogInput02;
	::DCS31_4:AI[1,3].RAW AT %IW."X20AI4322".AnalogInput03;
	::DCS31_4:AI[1,4].RAW AT %IW."X20AI4322".AnalogInput04;
	::DCS31_4:DI[1,5].In AT %IX."X20DI6371".DigitalInput05;
	::DCS31_4:DI[1,6].In AT %IX."X20DI6371".DigitalInput06;
END_VAR
```

## Configuration DCS34_1

CPU X20CP1584, AutomationRuntime C4.72, Build 4.1.2, Vc V4.72.0

### Task classes (Cpu.sw)
```
Cyclic#4:
  DCS34_1 <- DCS34_1.prg
Libraries: Lib489, standard, AsMbTCP, AsBrStr, asstring, operator, astime, AsIecCon, LibIP001, MTBasics, DRV_mbus, DataObj, sys_lib, brsystem, MTTypes, dvframe, runtime
```

### IoMap.iom - X20CP1584/IoMap.iom
```iecst
VAR_CONFIG
	::DCS34_1:AI[1,1].RAW AT %IW."X20AI8321".AnalogInput01;
	::DCS34_1:AI[1,2].RAW AT %IW."X20AI8321".AnalogInput02;
	::DCS34_1:AI[1,3].RAW AT %IW."X20AI8321".AnalogInput03;
	::DCS34_1:AI[1,4].RAW AT %IW."X20AI8321".AnalogInput04;
	::DCS34_1:AI[1,5].RAW AT %IW."X20AI8321".AnalogInput05;
	::DCS34_1:AI[1,6].RAW AT %IW."X20AI8321".AnalogInput06;
	::DCS34_1:AI[1,7].RAW AT %IW."X20AI8321".AnalogInput07;
	::DCS34_1:AI[1,8].RAW AT %IW."X20AI8321".AnalogInput08;
	::DCS34_1:AO[1,1].RAW AT %QW."X20AO2622".AnalogOutput01;
	::DCS34_1:DI[1,1].In AT %IX."X20DI8371".DigitalInput01;
	::DCS34_1:DI[1,2].In AT %IX."X20DI8371".DigitalInput02;
	::DCS34_1:DI[1,3].In AT %IX."X20DI8371".DigitalInput03;
	::DCS34_1:DI[1,4].In AT %IX."X20DI8371".DigitalInput04;
	::DCS34_1:DO_[1,1].Out AT %QX."X20DO6322".DigitalOutput01;
	::DCS34_1:DO_[1,2].Out AT %QX."X20DO6322".DigitalOutput02;
	::DCS34_1:DO_[1,3].Out AT %QX."X20DO6322".DigitalOutput03;
	::DCS34_1:DO_[1,4].Out AT %QX."X20DO6322".DigitalOutput04;
	::DCS34_1:DO_[1,5].Out AT %QX."X20DO6322".DigitalOutput05;
	::DCS34_1:DO_[1,6].Out AT %QX."X20DO6322".DigitalOutput06;
	::DCS34_1:AO[1,2].RAW AT %QW."X20AO2622".AnalogOutput02;
	::DCS34_1:DI[1,5].In AT %IX."X20DI8371".DigitalInput05;
	::DCS34_1:DI[1,6].In AT %IX."X20DI8371".DigitalInput06;
	::DCS34_1:DI[1,7].In AT %IX."X20DI8371".DigitalInput07;
	::DCS34_1:DI[1,8].In AT %IX."X20DI8371".DigitalInput08;
END_VAR
```

## Configuration DCS35_1

CPU X20CP0482, AutomationRuntime C4.72, Build 4.1.2, Vc V4.72.0

### Task classes (Cpu.sw)
```
Cyclic#4 (cycle 100000 us, tolerance 100000 us):
  DCS35_1 <- DCS35_1.prg
Libraries: Lib489, standard, AsMbTCP, AsBrStr, asstring, MTBasics, DRV_mbus, operator, astime, AsIecCon, LibIP001, DataObj, sys_lib, brsystem, MTTypes, dvframe, runtime
```

### Hardware
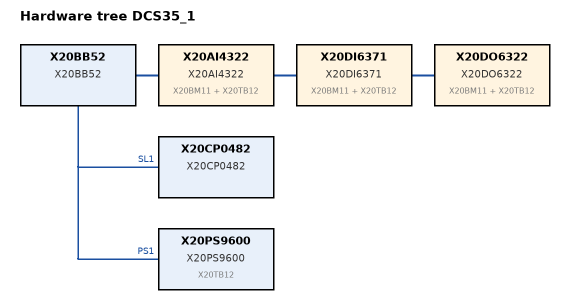
```
X20AI4322 : X20AI4322 v1.0.0.2  [SS1 -> X20TB12d.SS; SL -> X20BM11a.SL1]
X20BB52 : X20BB52 v1.1.0.0
X20BM11a : X20BM11 v1.0.0.1  [X2X1 -> X20BB52.IF6]
X20BM11b : X20BM11 v1.0.0.1  [X2X1 -> X20BM11a.X2X2]
X20BM11c : X20BM11 v1.0.0.1  [X2X1 -> X20BM11b.X2X2]
X20CP0482 : X20CP0482 v1.2.1.0  [SL -> X20BB52.SL1]
  Connector IF2:
    ActivateDevice = 1
    Mode = Manual
    InternetAddress = 192.168.50.18
    SubnetMask = 255.255.255.0
  ConfigurationID = IP001_DCS2_2
  TimerDeviceType = SWIOTIMER
  Cyclic1Duration = 10000
  Cyclic1Tolerance = 10000
  Cyclic2Duration = 20000
  Cyclic2Tolerance = 20000
  Cyclic3Duration = 50000
  Cyclic3Tolerance = 50000
  Cyclic4Duration = 100000
  Cyclic4Tolerance = 100000
  Cyclic5Duration = 200000
  Cyclic5Tolerance = 200000
  Cyclic6Duration = 500000
  Cyclic6Tolerance = 500000
  Cyclic7Duration = 1000000
  Cyclic7Tolerance = 1000000
  Cyclic8Duration = 10000
  Cyclic8Tolerance = 30000000
  ActivateOpcUa = 1
  OpcUa_AuthenticationSecurityPolicy_EnableNone = 1
  OpcUa_AuthenticationSecurityPolicy_EnableBasic128Rsa15 = 1
  OpcUaInformationModels_PV_Version = 1
X20DI6371 : X20DI6371 v1.0.2.0  [SS1 -> X20TB12b.SS; SL -> X20BM11b.SL1]
X20DO6322 : X20DO6322 v1.0.4.0  [SS1 -> X20TB12c.SS; SL -> X20BM11c.SL1]
X20PS9600 : X20PS9600 v1.0.2.0  [PS -> X20BB52.PS1; SS1 -> X20TB12.SS]
X20TB12 : X20TB12 v1.0.0.0
X20TB12b : X20TB12 v1.0.0.0
X20TB12c : X20TB12 v1.0.0.0
X20TB12d : X20TB12 v1.0.0.0
```

### IoMap.iom - X20CP0482/IoMap.iom
```iecst
VAR_CONFIG
	::DCS35_1:DI[1,1].In AT %IX."X20DI6371".DigitalInput01;
	::DCS35_1:DI[1,2].In AT %IX."X20DI6371".DigitalInput02;
	::DCS35_1:DI[1,3].In AT %IX."X20DI6371".DigitalInput03;
	::DCS35_1:DI[1,4].In AT %IX."X20DI6371".DigitalInput04;
	::DCS35_1:DO_[1,1].Out AT %QX."X20DO6322".DigitalOutput01;
	::DCS35_1:DO_[1,2].Out AT %QX."X20DO6322".DigitalOutput02;
	::DCS35_1:DO_[1,3].Out AT %QX."X20DO6322".DigitalOutput03;
	::DCS35_1:DO_[1,4].Out AT %QX."X20DO6322".DigitalOutput04;
	::DCS35_1:AI[1,1].RAW AT %IW."X20AI4322".AnalogInput01;
	::DCS35_1:AI[1,2].RAW AT %IW."X20AI4322".AnalogInput02;
	::DCS35_1:AI[1,3].RAW AT %IW."X20AI4322".AnalogInput03;
	::DCS35_1:AI[1,4].RAW AT %IW."X20AI4322".AnalogInput04;
	::DCS35_1:DI[1,5].In AT %IX."X20DI6371".DigitalInput05;
	::DCS35_1:DI[1,6].In AT %IX."X20DI6371".DigitalInput06;
	::DCS35_1:DO_[1,5].Out  AT %QX."X20DO6322".DigitalOutput05;
	::DCS35_1:DO_[1,6].Out  AT %QX."X20DO6322".DigitalOutput06;
END_VAR
```

## Configuration DCS36_1

CPU X20CP0482, AutomationRuntime C4.72, Build 4.1.2, Vc V4.72.0

### Task classes (Cpu.sw)
```
Cyclic#4 (cycle 100000 us, tolerance 100000 us):
  DCS36_1 <- DCS36_1.prg
Libraries: Lib489, standard, AsMbTCP, operator, astime, AsIecCon, LibIP001, AsBrStr, asstring, MTBasics, DRV_mbus, DataObj, sys_lib, brsystem, MTTypes, dvframe, runtime
```

### Hardware
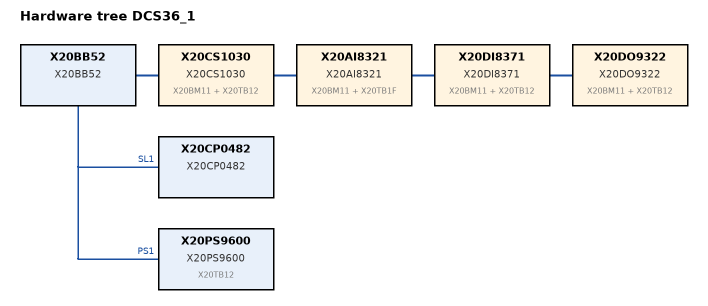
```
X20AI8321 : X20AI8321 v1.4.0.0  [SS1 -> X20TB1F.SS; SL -> X20BM11a.SL1]
X20BB52 : X20BB52 v1.1.0.0
X20BM11 : X20BM11 v1.0.0.1  [X2X1 -> X20BB52.IF6]
X20BM11a : X20BM11 v1.0.0.1  [X2X1 -> X20BM11.X2X2]
X20BM11b : X20BM11 v1.0.0.1  [X2X1 -> X20BM11a.X2X2]
X20BM11c : X20BM11 v1.0.0.1  [X2X1 -> X20BM11b.X2X2]
X20CP0482 : X20CP0482 v1.2.1.0  [SL -> X20BB52.SL1]
  Connector IF2:
    ActivateDevice = 1
    Mode = Manual
    InternetAddress = 192.168.50.18
    SubnetMask = 255.255.255.0
  ConfigurationID = IP001_DCS2_2
  TimerDeviceType = SWIOTIMER
  Cyclic1Duration = 10000
  Cyclic1Tolerance = 10000
  Cyclic2Duration = 20000
  Cyclic2Tolerance = 20000
  Cyclic3Duration = 50000
  Cyclic3Tolerance = 50000
  Cyclic4Duration = 100000
  Cyclic4Tolerance = 100000
  Cyclic5Duration = 200000
  Cyclic5Tolerance = 200000
  Cyclic6Duration = 500000
  Cyclic6Tolerance = 500000
  Cyclic7Duration = 1000000
  Cyclic7Tolerance = 1000000
  Cyclic8Duration = 10000
  Cyclic8Tolerance = 30000000
  ActivateOpcUa = 1
  OpcUa_AuthenticationSecurityPolicy_EnableNone = 1
  OpcUa_AuthenticationSecurityPolicy_EnableBasic128Rsa15 = 1
  OpcUaInformationModels_PV_Version = 1
X20CS1030 : X20CS1030 v1.7.0.0  [SS1 -> X20TB12a.SS; SL -> X20BM11.SL1]
X20DI8371 : X20DI8371 v1.0.2.0  [SS1 -> X20TB12b.SS; SL -> X20BM11b.SL1]
X20DO9322 : X20DO9322 v1.1.0.0  [SS1 -> X20TB12c.SS; SL -> X20BM11c.SL1]
X20PS9600 : X20PS9600 v1.0.2.0  [PS -> X20BB52.PS1; SS1 -> X20TB12.SS]
X20TB12 : X20TB12 v1.0.0.0
X20TB12a : X20TB12 v1.0.0.0
X20TB12b : X20TB12 v1.0.0.0
X20TB12c : X20TB12 v1.0.0.0
X20TB1F : X20TB1F v1.0.0.0
```

### IoMap.iom - X20CP0482/IoMap.iom
```iecst
VAR_CONFIG
	::DCS36_1:DI[1,1].In AT %IX."X20DI8371".DigitalInput01;
	::DCS36_1:DI[1,2].In AT %IX."X20DI8371".DigitalInput02;
	::DCS36_1:DI[1,3].In AT %IX."X20DI8371".DigitalInput03;
	::DCS36_1:DI[1,4].In AT %IX."X20DI8371".DigitalInput04;
	::DCS36_1:DO_[1,1].Out AT %QX."X20DO9322".DigitalOutput01;
	::DCS36_1:DO_[1,2].Out AT %QX."X20DO9322".DigitalOutput02;
	::DCS36_1:DO_[1,3].Out AT %QX."X20DO9322".DigitalOutput03;
	::DCS36_1:DO_[1,4].Out AT %QX."X20DO9322".DigitalOutput04;
	::DCS36_1:AI[1,1].RAW AT %IW."X20AI8321".AnalogInput01;
	::DCS36_1:AI[1,2].RAW AT %IW."X20AI8321".AnalogInput02;
	::DCS36_1:AI[1,3].RAW AT %IW."X20AI8321".AnalogInput03;
	::DCS36_1:AI[1,4].RAW AT %IW."X20AI8321".AnalogInput04;
	::DCS36_1:DI[1,5].In AT %IX."X20DI8371".DigitalInput05;
	::DCS36_1:DI[1,6].In AT %IX."X20DI8371".DigitalInput06;
	::DCS36_1:AI[1,5].RAW AT %IW."X20AI8321".AnalogInput05;
	::DCS36_1:AI[1,6].RAW AT %IW."X20AI8321".AnalogInput06;
	::DCS36_1:AI[1,7].RAW AT %IW."X20AI8321".AnalogInput07;
	::DCS36_1:AI[1,8].RAW AT %IW."X20AI8321".AnalogInput08;
	::DCS36_1:DI[1,7].In AT %IX."X20DI8371".DigitalInput07;
	::DCS36_1:DI[1,8].In AT %IX."X20DI8371".DigitalInput08;
	::DCS36_1:DO_[1,5].Out AT %QX."X20DO9322".DigitalOutput05;
	::DCS36_1:DO_[1,6].Out AT %QX."X20DO9322".DigitalOutput06;
	::DCS36_1:DO_[1,7].Out  AT %QX."X20DO9322".DigitalOutput07;
	::DCS36_1:DO_[1,8].Out AT %QX."X20DO9322".DigitalOutput08;
	::DCS36_1:DO_[1,9].Out AT %QX."X20DO9322".DigitalOutput09;
	::DCS36_1:DO_[1,10].Out AT %QX."X20DO9322".DigitalOutput10;
	::DCS36_1:DO_[1,11].Out AT %QX."X20DO9322".DigitalOutput11;
	::DCS36_1:DO_[1,12].Out AT %QX."X20DO9322".DigitalOutput12;
END_VAR
```

## Configuration DCS37_1

### Task classes (Cpu.sw)
```
Cyclic#4 (cycle 100000 us, tolerance 100000 us):
  DCS37_1 <- DCS37_1.prg
Libraries: Lib489, standard, AsMbTCP, AsBrStr, asstring, MTBasics, DRV_mbus, DataObj, sys_lib, brsystem, MTTypes, dvframe, runtime
```

### Hardware
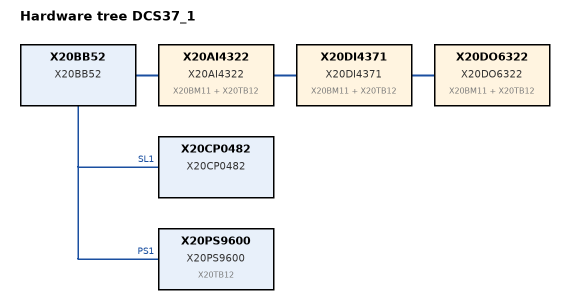
```
X20AI4322 : X20AI4322 v1.0.0.2  [SS1 -> X20TB12d.SS; SL -> X20BM11a.SL1]
X20BB52 : X20BB52 v1.1.0.0
X20BM11a : X20BM11 v1.0.0.1  [X2X1 -> X20BB52.IF6]
X20BM11b : X20BM11 v1.0.0.1  [X2X1 -> X20BM11a.X2X2]
X20BM11c : X20BM11 v1.0.0.1  [X2X1 -> X20BM11b.X2X2]
X20CP0482 : X20CP0482 v1.2.1.0  [SL -> X20BB52.SL1]
  Connector IF2:
    ActivateDevice = 1
    Mode = Manual
    InternetAddress = 192.168.50.18
    SubnetMask = 255.255.255.0
  ConfigurationID = IP001_DCS2_2
  TimerDeviceType = SWIOTIMER
  Cyclic1Duration = 10000
  Cyclic1Tolerance = 10000
  Cyclic2Duration = 20000
  Cyclic2Tolerance = 20000
  Cyclic3Duration = 50000
  Cyclic3Tolerance = 50000
  Cyclic4Duration = 100000
  Cyclic4Tolerance = 100000
  Cyclic5Duration = 200000
  Cyclic5Tolerance = 200000
  Cyclic6Duration = 500000
  Cyclic6Tolerance = 500000
  Cyclic7Duration = 1000000
  Cyclic7Tolerance = 1000000
  Cyclic8Duration = 10000
  Cyclic8Tolerance = 30000000
  ActivateOpcUa = 1
  OpcUa_AuthenticationSecurityPolicy_EnableNone = 1
  OpcUa_AuthenticationSecurityPolicy_EnableBasic128Rsa15 = 1
  OpcUaInformationModels_PV_Version = 1
X20DI4371 : X20DI4371 v1.0.3.0  [SS1 -> X20TB12b.SS; SL -> X20BM11b.SL1]
X20DO6322 : X20DO6322 v1.0.4.0  [SS1 -> X20TB12c.SS; SL -> X20BM11c.SL1]
X20PS9600 : X20PS9600 v1.0.2.0  [PS -> X20BB52.PS1; SS1 -> X20TB12.SS]
X20TB12 : X20TB12 v1.0.0.0
X20TB12b : X20TB12 v1.0.0.0
X20TB12c : X20TB12 v1.0.0.0
X20TB12d : X20TB12 v1.0.0.0
```

### IoMap.iom - X20CP0482/IoMap.iom
```iecst
VAR_CONFIG
	::DCS37_1:DI[1,1].In AT %IX."X20DI4371".DigitalInput01;
	::DCS37_1:DI[1,2].In AT %IX."X20DI4371".DigitalInput02;
	::DCS37_1:DI[1,3].In AT %IX."X20DI4371".DigitalInput03;
	::DCS37_1:DI[1,4].In AT %IX."X20DI4371".DigitalInput04;
	::DCS37_1:DO_[1,1].Out AT %QX."X20DO6322".DigitalOutput01;
	::DCS37_1:DO_[1,2].Out AT %QX."X20DO6322".DigitalOutput02;
	::DCS37_1:DO_[1,3].Out AT %QX."X20DO6322".DigitalOutput03;
	::DCS37_1:DO_[1,4].Out AT %QX."X20DO6322".DigitalOutput04;
	::DCS37_1:AI[1,1].RAW AT %IW."X20AI4322".AnalogInput01;
	::DCS37_1:AI[1,2].RAW AT %IW."X20AI4322".AnalogInput02;
	::DCS37_1:AI[1,3].RAW AT %IW."X20AI4322".AnalogInput03;
	::DCS37_1:AI[1,4].RAW AT %IW."X20AI4322".AnalogInput04;
	::DCS37_1:DO_[1,5].Out AT %QX."X20DO6322".DigitalOutput05;
	::DCS37_1:DO_[1,6].Out AT %QX."X20DO6322".DigitalOutput06;
END_VAR
```

## Configuration DCS39_1

### Task classes (Cpu.sw)
```
Cyclic#4:
  DCS39_1 <- DCS39_1.prg
Libraries: Lib489, standard, AsMbTCP, AsBrStr, operator, astime, AsIecCon, LibIP001, asstring, MTBasics, DRV_mbus, DataObj, sys_lib, brsystem, MTTypes, dvframe, runtime
```

### IoMap.iom - X20CP1584/IoMap.iom
```iecst
VAR_CONFIG
	::DCS39_1:AI[1,1].RAW AT %IW."X20AI8321".AnalogInput01;
	::DCS39_1:AI[1,2].RAW AT %IW."X20AI8321".AnalogInput02;
	::DCS39_1:AI[1,3].RAW AT %IW."X20AI8321".AnalogInput03;
	::DCS39_1:AI[1,4].RAW AT %IW."X20AI8321".AnalogInput04;
	::DCS39_1:AI[1,5].RAW AT %IW."X20AI8321".AnalogInput05;
	::DCS39_1:AI[1,6].RAW AT %IW."X20AI8321".AnalogInput06;
	::DCS39_1:AI[1,7].RAW AT %IW."X20AI8321".AnalogInput07;
	::DCS39_1:AI[1,8].RAW AT %IW."X20AI8321".AnalogInput08;
	::DCS39_1:AO[1,1].RAW AT %QW."X20AO2622".AnalogOutput01;
	::DCS39_1:DI[1,1].In AT %IX."X20DI8371".DigitalInput01;
	::DCS39_1:DI[1,2].In AT %IX."X20DI8371".DigitalInput02;
	::DCS39_1:DI[1,3].In AT %IX."X20DI8371".DigitalInput03;
	::DCS39_1:DI[1,4].In AT %IX."X20DI8371".DigitalInput04;
	::DCS39_1:DO_[1,1].Out AT %QX."X20DO6322".DigitalOutput01;
	::DCS39_1:DO_[1,2].Out AT %QX."X20DO6322".DigitalOutput02;
	::DCS39_1:DO_[1,3].Out AT %QX."X20DO6322".DigitalOutput03;
	::DCS39_1:DO_[1,4].Out AT %QX."X20DO6322".DigitalOutput04;
	::DCS39_1:DO_[1,5].Out AT %QX."X20DO6322".DigitalOutput05;
	::DCS39_1:DO_[1,6].Out AT %QX."X20DO6322".DigitalOutput06;
	::DCS39_1:AO[1,2].RAW AT %QW."X20AO2622".AnalogOutput02;
	::DCS39_1:DI[1,5].In AT %IX."X20DI8371".DigitalInput05;
	::DCS39_1:DI[1,6].In AT %IX."X20DI8371".DigitalInput06;
	::DCS39_1:DI[1,7].In AT %IX."X20DI8371".DigitalInput07;
	::DCS39_1:DI[1,8].In AT %IX."X20DI8371".DigitalInput08;
END_VAR
```

## Configuration DCS40_1

### Task classes (Cpu.sw)
```
Cyclic#4:
  DCS40_1 <- DCS40_1.prg
Binaries: FWRules, udbdef, TCData, arconfig, User, Role, iomap, asfw, ashwac, ashwd, sysconf
Libraries: Lib489, standard, AsMbTCP, AsBrStr, asstring, MTBasics, operator, astime, AsIecCon, LibIP001, DRV_mbus, DataObj, sys_lib, brsystem, MTTypes, dvframe, runtime
```

### Hardware
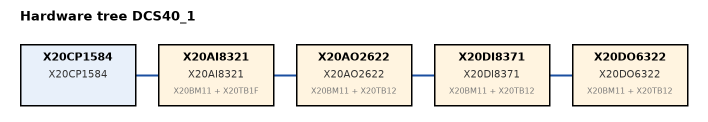
```
X20AI8321 : X20AI8321 v1.4.0.0  [SS1 -> X20TB1F.SS; SL -> X20BM11a.SL1]
X20AO2622 : X20AO2622 v1.1.0.0  [SS1 -> X20TB12e.SS; SL -> X20BM11e.SL1]
X20BM11a : X20BM11 v1.0.0.1  [X2X1 -> X20CP1584.IF6]
X20BM11b : X20BM11 v1.0.0.1  [X2X1 -> X20BM11e.X2X2]
X20BM11c : X20BM11 v1.0.0.1  [X2X1 -> X20BM11b.X2X2]
X20BM11e : X20BM11 v1.0.0.1  [X2X1 -> X20BM11a.X2X2]
X20CP1584 : X20CP1584 v1.8.0.0
  Connector IF2:
    ActivateDevice = 1
    Mode = Manual
    InternetAddress = 192.168.50.13
    SubnetMask = 255.255.255.0
  ConfigurationID = IP001_DCS2_2
  ActivateOpcUa = 1
  OpcUa_AuthenticationSecurityPolicy_EnableNone = 1
  OpcUa_AuthenticationSecurityPolicy_EnableBasic128Rsa15 = 1
  OpcUaInformationModels_PV_Version = 1
X20DI8371 : X20DI8371 v1.0.2.0  [SS1 -> X20TB12.SS; SL -> X20BM11b.SL1]
X20DO6322 : X20DO6322 v1.0.4.0  [SS1 -> X20TB12c.SS; SL -> X20BM11c.SL1]
X20TB12 : X20TB12 v1.0.0.0
X20TB12c : X20TB12 v1.0.0.0
X20TB12e : X20TB12 v1.0.0.0
X20TB1F : X20TB1F v1.0.0.0
```

### IoMap.iom - X20CP1584/IoMap.iom
```iecst
VAR_CONFIG
	::DCS40_1:AI[1,1].RAW AT %IW."X20AI8321".AnalogInput01;
	::DCS40_1:AI[1,2].RAW AT %IW."X20AI8321".AnalogInput02;
	::DCS40_1:AI[1,3].RAW AT %IW."X20AI8321".AnalogInput03;
	::DCS40_1:AI[1,4].RAW AT %IW."X20AI8321".AnalogInput04;
	::DCS40_1:AI[1,5].RAW AT %IW."X20AI8321".AnalogInput05;
	::DCS40_1:AI[1,6].RAW AT %IW."X20AI8321".AnalogInput06;
	::DCS40_1:AI[1,7].RAW AT %IW."X20AI8321".AnalogInput07;
	::DCS40_1:AI[1,8].RAW AT %IW."X20AI8321".AnalogInput08;
	::DCS40_1:AO[1,1].RAW AT %QW."X20AO2622".AnalogOutput01;
	::DCS40_1:DI[1,1].In AT %IX."X20DI8371".DigitalInput01;
	::DCS40_1:DI[1,2].In AT %IX."X20DI8371".DigitalInput02;
	::DCS40_1:DI[1,3].In AT %IX."X20DI8371".DigitalInput03;
	::DCS40_1:DI[1,4].In AT %IX."X20DI8371".DigitalInput04;
	::DCS40_1:DO_[1,1].Out AT %QX."X20DO6322".DigitalOutput01;
	::DCS40_1:DO_[1,2].Out AT %QX."X20DO6322".DigitalOutput02;
	::DCS40_1:DO_[1,3].Out AT %QX."X20DO6322".DigitalOutput03;
	::DCS40_1:DO_[1,4].Out AT %QX."X20DO6322".DigitalOutput04;
	::DCS40_1:DO_[1,5].Out AT %QX."X20DO6322".DigitalOutput05;
	::DCS40_1:DO_[1,6].Out AT %QX."X20DO6322".DigitalOutput06;
	::DCS40_1:AO[1,2].RAW AT %QW."X20AO2622".AnalogOutput02;
	::DCS40_1:DI[1,5].In AT %IX."X20DI8371".DigitalInput05;
	::DCS40_1:DI[1,6].In AT %IX."X20DI8371".DigitalInput06;
	::DCS40_1:DI[1,7].In AT %IX."X20DI8371".DigitalInput07;
	::DCS40_1:DI[1,8].In AT %IX."X20DI8371".DigitalInput08;
END_VAR
```

## Configuration DCS45_1

### Hardware
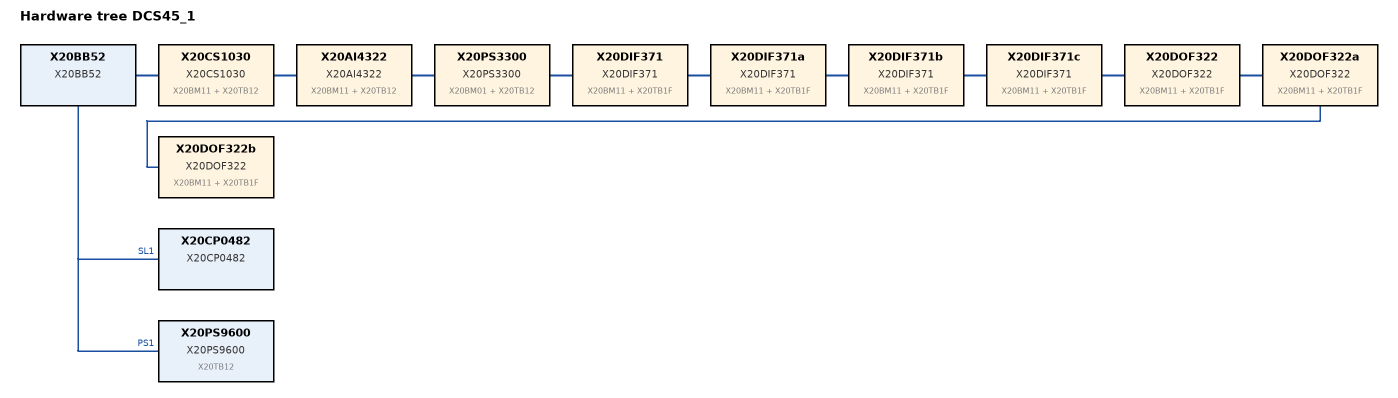
```
X20AI4322 : X20AI4322 v1.0.0.2  [SS1 -> X20TB12c.SS; SL -> X20BM11d.SL1]
X20BB52 : X20BB52 v1.1.0.0
X20BM01 : X20BM01 v2.1.0.0  [X2X1 -> X20BM11d.X2X2]
X20BM11 : X20BM11 v1.0.0.1  [X2X1 -> X20BB52.IF6]
X20BM11b : X20BM11 v1.0.0.1  [X2X1 -> X20BM01.X2X2]
X20BM11c : X20BM11 v1.0.0.1  [X2X1 -> X20BM11k.X2X2]
X20BM11d : X20BM11 v1.0.0.1  [X2X1 -> X20BM11.X2X2]
X20BM11e : X20BM11 v1.0.0.1  [X2X1 -> X20BM11b.X2X2]
X20BM11j : X20BM11 v1.0.0.1  [X2X1 -> X20BM11e.X2X2]
X20BM11k : X20BM11 v1.0.0.1  [X2X1 -> X20BM11j.X2X2]
X20BM11p : X20BM11 v1.0.0.1  [X2X1 -> X20BM11c.X2X2]
X20BM11q : X20BM11 v1.0.0.1  [X2X1 -> X20BM11p.X2X2]
X20CP0482 : X20CP0482 v1.2.1.0  [SL -> X20BB52.SL1]
  Connector IF2:
    ActivateDevice = 1
    Mode = Manual
    InternetAddress = 192.168.50.28
    SubnetMask = 255.255.255.0
  ConfigurationID = IP001_DCS45_1
  TimerDeviceType = SWIOTIMER
  Cyclic1Duration = 10000
  Cyclic1Tolerance = 10000
  Cyclic2Duration = 20000
  Cyclic2Tolerance = 20000
  Cyclic3Duration = 50000
  Cyclic3Tolerance = 50000
  Cyclic4Duration = 100000
  Cyclic4Tolerance = 100000
  Cyclic5Duration = 200000
  Cyclic5Tolerance = 200000
  Cyclic6Duration = 500000
  Cyclic6Tolerance = 500000
  Cyclic7Duration = 1000000
  Cyclic7Tolerance = 1000000
  Cyclic8Duration = 10000
  Cyclic8Tolerance = 30000000
  ActivateOpcUa = 1
  OpcUa_AuthenticationSecurityPolicy_EnableNone = 1
  OpcUa_AuthenticationSecurityPolicy_EnableBasic128Rsa15 = 1
  OpcUaInformationModels_PV_Version = 1
X20CS1030 : X20CS1030 v1.7.0.0  [SS1 -> X20TB12b.SS; SL -> X20BM11.SL1]
X20DIF371 : X20DIF371 v1.1.0.0  [SS1 -> X20TB1F6.SS; SL -> X20BM11b.SL1]
X20DIF371a : X20DIF371 v1.1.0.0  [SS1 -> X20TB1F7.SS; SL -> X20BM11e.SL1]
X20DIF371b : X20DIF371 v1.1.0.0  [SS1 -> X20TB1F8.SS; SL -> X20BM11j.SL1]
X20DIF371c : X20DIF371 v1.1.0.0  [SS1 -> X20TB1F9.SS; SL -> X20BM11k.SL1]
X20DOF322 : X20DOF322 v1.4.0.0  [SS1 -> X20TB1F14.SS; SL -> X20BM11c.SL1]
X20DOF322a : X20DOF322 v1.4.0.0  [SS1 -> X20TB1F15.SS; SL -> X20BM11p.SL1]
X20DOF322b : X20DOF322 v1.4.0.0  [SS1 -> X20TB1F16.SS; SL -> X20BM11q.SL1]
X20PS3300 : X20PS3300 v1.1.0.0  [SS1 -> X20TB12.SS; SL -> X20BM01.SL1]
X20PS9600 : X20PS9600 v1.0.2.0  [PS -> X20BB52.PS1; SS1 -> X20TB12a.SS]
X20TB12 : X20TB12 v1.0.0.0
X20TB12a : X20TB12 v1.0.0.0
X20TB12b : X20TB12 v1.0.0.0
X20TB12c : X20TB12 v1.0.0.0
X20TB1F14 : X20TB1F v1.0.0.0
X20TB1F15 : X20TB1F v1.0.0.0
X20TB1F16 : X20TB1F v1.0.0.0
X20TB1F6 : X20TB1F v1.0.0.0
X20TB1F7 : X20TB1F v1.0.0.0
X20TB1F8 : X20TB1F v1.0.0.0
X20TB1F9 : X20TB1F v1.0.0.0
```

### IoMap.iom - X20CP0482/IoMap.iom
```iecst
VAR_CONFIG
	::DCS45_1:DI[1,1].In AT %IX."X20DIF371".DigitalInput01;
	::DCS45_1:DI[1,2].In AT %IX."X20DIF371".DigitalInput02;
	::DCS45_1:DI[1,3].In AT %IX."X20DIF371".DigitalInput03;
	::DCS45_1:DI[1,4].In AT %IX."X20DIF371".DigitalInput04;
	::DCS45_1:DI[1,5].In AT %IX."X20DIF371".DigitalInput05;
	::DCS45_1:DI[1,6].In AT %IX."X20DIF371".DigitalInput06;
	::DCS45_1:DI[1,7].In AT %IX."X20DIF371".DigitalInput07;
	::DCS45_1:DI[1,8].In AT %IX."X20DIF371".DigitalInput08;
	::DCS45_1:DI[1,9].In AT %IX."X20DIF371".DigitalInput09;
	::DCS45_1:DI[1,10].In AT %IX."X20DIF371".DigitalInput10;
	::DCS45_1:DI[1,11].In AT %IX."X20DIF371".DigitalInput11;
	::DCS45_1:DI[1,12].In AT %IX."X20DIF371".DigitalInput12;
	::DCS45_1:DI[1,13].In AT %IX."X20DIF371".DigitalInput13;
	::DCS45_1:DI[1,14].In AT %IX."X20DIF371".DigitalInput14;
	::DCS45_1:DI[1,15].In AT %IX."X20DIF371".DigitalInput15;
	::DCS45_1:DI[1,16].In AT %IX."X20DIF371".DigitalInput16;
	::DCS45_1:DI[2,1].In AT %IX."X20DIF371a".DigitalInput01;
	::DCS45_1:DI[2,2].In AT %IX."X20DIF371a".DigitalInput02;
	::DCS45_1:DI[2,3].In AT %IX."X20DIF371a".DigitalInput03;
	::DCS45_1:DI[2,4].In AT %IX."X20DIF371a".DigitalInput04;
	::DCS45_1:DI[2,5].In AT %IX."X20DIF371a".DigitalInput05;
	::DCS45_1:DI[2,6].In AT %IX."X20DIF371a".DigitalInput06;
	::DCS45_1:DI[2,7].In AT %IX."X20DIF371a".DigitalInput07;
	::DCS45_1:DI[2,8].In AT %IX."X20DIF371a".DigitalInput08;
	::DCS45_1:DI[2,9].In AT %IX."X20DIF371a".DigitalInput09;
	::DCS45_1:DI[2,10].In AT %IX."X20DIF371a".DigitalInput10;
	::DCS45_1:DI[2,11].In AT %IX."X20DIF371a".DigitalInput11;
	::DCS45_1:DI[2,12].In AT %IX."X20DIF371a".DigitalInput12;
	::DCS45_1:DI[2,13].In AT %IX."X20DIF371a".DigitalInput13;
	::DCS45_1:DI[2,14].In AT %IX."X20DIF371a".DigitalInput14;
	::DCS45_1:DI[2,15].In AT %IX."X20DIF371a".DigitalInput15;
	::DCS45_1:DI[2,16].In AT %IX."X20DIF371a".DigitalInput16;
	::DCS45_1:DI[3,1].In AT %IX."X20DIF371b".DigitalInput01;
	::DCS45_1:DI[3,2].In AT %IX."X20DIF371b".DigitalInput02;
	::DCS45_1:DI[3,3].In AT %IX."X20DIF371b".DigitalInput03;
	::DCS45_1:DI[3,4].In AT %IX."X20DIF371b".DigitalInput04;
	::DCS45_1:DI[3,5].In AT %IX."X20DIF371b".DigitalInput05;
	::DCS45_1:DI[3,6].In AT %IX."X20DIF371b".DigitalInput06;
	::DCS45_1:DI[3,7].In AT %IX."X20DIF371b".DigitalInput07;
	::DCS45_1:DI[3,8].In AT %IX."X20DIF371b".DigitalInput08;
	::DCS45_1:DI[3,9].In AT %IX."X20DIF371b".DigitalInput09;
	::DCS45_1:DI[3,10].In AT %IX."X20DIF371b".DigitalInput10;
	::DCS45_1:DI[3,11].In AT %IX."X20DIF371b".DigitalInput11;
	::DCS45_1:DI[3,12].In AT %IX."X20DIF371b".DigitalInput12;
	::DCS45_1:DI[3,13].In AT %IX."X20DIF371b".DigitalInput13;
	::DCS45_1:DI[3,14].In AT %IX."X20DIF371b".DigitalInput14;
	::DCS45_1:DI[3,15].In AT %IX."X20DIF371b".DigitalInput15;
	::DCS45_1:DI[3,16].In AT %IX."X20DIF371b".DigitalInput16;
	::DCS45_1:DI[4,1].In AT %IX."X20DIF371c".DigitalInput01;
	::DCS45_1:DI[4,2].In AT %IX."X20DIF371c".DigitalInput02;
	::DCS45_1:DI[4,3].In AT %IX."X20DIF371c".DigitalInput03;
	::DCS45_1:DI[4,4].In AT %IX."X20DIF371c".DigitalInput04;
	::DCS45_1:DI[4,5].In AT %IX."X20DIF371c".DigitalInput05;
	::DCS45_1:DI[4,6].In AT %IX."X20DIF371c".DigitalInput06;
	::DCS45_1:DI[4,7].In AT %IX."X20DIF371c".DigitalInput07;
	::DCS45_1:DI[4,8].In AT %IX."X20DIF371c".DigitalInput08;
	::DCS45_1:DI[4,9].In AT %IX."X20DIF371c".DigitalInput09;
	::DCS45_1:DI[4,10].In AT %IX."X20DIF371c".DigitalInput10;
	::DCS45_1:DI[4,11].In AT %IX."X20DIF371c".DigitalInput11;
	::DCS45_1:DI[4,12].In AT %IX."X20DIF371c".DigitalInput12;
	::DCS45_1:DI[4,13].In AT %IX."X20DIF371c".DigitalInput13;
	::DCS45_1:DI[4,14].In AT %IX."X20DIF371c".DigitalInput14;
	::DCS45_1:DI[4,15].In AT %IX."X20DIF371c".DigitalInput15;
	::DCS45_1:DI[4,16].In AT %IX."X20DIF371c".DigitalInput16;
	::DCS45_1:DO_[1,1].Out AT %QX."X20DOF322".DigitalOutput01;
	::DCS45_1:DO_[1,2].Out AT %QX."X20DOF322".DigitalOutput02;
	::DCS45_1:DO_[1,3].Out AT %QX."X20DOF322".DigitalOutput03;
	::DCS45_1:DO_[1,4].Out AT %QX."X20DOF322".DigitalOutput04;
	::DCS45_1:DO_[1,5].Out AT %QX."X20DOF322".DigitalOutput05;
	::DCS45_1:DO_[1,6].Out AT %QX."X20DOF322".DigitalOutput06;
	::DCS45_1:DO_[1,7].Out AT %QX."X20DOF322".DigitalOutput07;
	::DCS45_1:DO_[1,8].Out AT %QX."X20DOF322".DigitalOutput08;
	::DCS45_1:DO_[1,9].Out AT %QX."X20DOF322".DigitalOutput09;
	::DCS45_1:DO_[1,10].Out AT %QX."X20DOF322".DigitalOutput10;
	::DCS45_1:DO_[1,11].Out AT %QX."X20DOF322".DigitalOutput11;
	::DCS45_1:DO_[1,12].Out AT %QX."X20DOF322".DigitalOutput12;
	::DCS45_1:DO_[1,13].Out AT %QX."X20DOF322".DigitalOutput13;
	::DCS45_1:DO_[1,14].Out AT %QX."X20DOF322".DigitalOutput14;
	::DCS45_1:DO_[1,15].Out AT %QX."X20DOF322".DigitalOutput15;
	::DCS45_1:DO_[1,16].Out AT %QX."X20DOF322".DigitalOutput16;
	::DCS45_1:DO_[2,1].Out AT %QX."X20DOF322a".DigitalOutput01;
	::DCS45_1:DO_[2,2].Out AT %QX."X20DOF322a".DigitalOutput02;
	::DCS45_1:DO_[2,3].Out AT %QX."X20DOF322a".DigitalOutput03;
	::DCS45_1:DO_[2,4].Out AT %QX."X20DOF322a".DigitalOutput04;
	::DCS45_1:DO_[2,5].Out AT %QX."X20DOF322a".DigitalOutput05;
	::DCS45_1:DO_[2,6].Out AT %QX."X20DOF322a".DigitalOutput06;
	::DCS45_1:DO_[2,7].Out AT %QX."X20DOF322a".DigitalOutput07;
	::DCS45_1:DO_[2,8].Out AT %QX."X20DOF322a".DigitalOutput08;
	::DCS45_1:DO_[2,9].Out AT %QX."X20DOF322a".DigitalOutput09;
	::DCS45_1:DO_[2,10].Out AT %QX."X20DOF322a".DigitalOutput10;
	::DCS45_1:DO_[2,11].Out AT %QX."X20DOF322a".DigitalOutput11;
	::DCS45_1:DO_[2,12].Out AT %QX."X20DOF322a".DigitalOutput12;
	::DCS45_1:DO_[2,13].Out AT %QX."X20DOF322a".DigitalOutput13;
	::DCS45_1:DO_[2,14].Out AT %QX."X20DOF322a".DigitalOutput14;
	::DCS45_1:DO_[2,15].Out AT %QX."X20DOF322a".DigitalOutput15;
	::DCS45_1:DO_[2,16].Out AT %QX."X20DOF322a".DigitalOutput16;
	::DCS45_1:DO_[3,1].Out AT %QX."X20DOF322b".DigitalOutput01;
	::DCS45_1:DO_[3,2].Out AT %QX."X20DOF322b".DigitalOutput02;
	::DCS45_1:DO_[3,3].Out AT %QX."X20DOF322b".DigitalOutput03;
	::DCS45_1:DO_[3,4].Out AT %QX."X20DOF322b".DigitalOutput04;
	::DCS45_1:DO_[3,5].Out AT %QX."X20DOF322b".DigitalOutput05;
	::DCS45_1:DO_[3,6].Out AT %QX."X20DOF322b".DigitalOutput06;
	::DCS45_1:DO_[3,7].Out AT %QX."X20DOF322b".DigitalOutput07;
	::DCS45_1:DO_[3,8].Out AT %QX."X20DOF322b".DigitalOutput08;
	::DCS45_1:DO_[3,9].Out AT %QX."X20DOF322b".DigitalOutput09;
	::DCS45_1:DO_[3,10].Out AT %QX."X20DOF322b".DigitalOutput10;
	::DCS45_1:DO_[3,11].Out AT %QX."X20DOF322b".DigitalOutput11;
	::DCS45_1:DO_[3,12].Out AT %QX."X20DOF322b".DigitalOutput12;
	::DCS45_1:DO_[3,13].Out AT %QX."X20DOF322b".DigitalOutput13;
	::DCS45_1:DO_[3,14].Out AT %QX."X20DOF322b".DigitalOutput14;
	::DCS45_1:DO_[3,15].Out AT %QX."X20DOF322b".DigitalOutput15;
	::DCS45_1:DO_[3,16].Out AT %QX."X20DOF322b".DigitalOutput16;
	::DCS45_1:AI[1,1].RAW AT %IW."X20AI4322".AnalogInput01;
	::DCS45_1:AI[1,2].RAW AT %IW."X20AI4322".AnalogInput02;
	::DCS45_1:AI[1,3].RAW AT %IW."X20AI4322".AnalogInput03;
	::DCS45_1:AI[1,4].RAW AT %IW."X20AI4322".AnalogInput04;
END_VAR
```

## Configuration DCS4_1

CPU X20CP1584, AutomationRuntime B4.92, Build 4.1.2, Vc V4.72.5

### Hardware
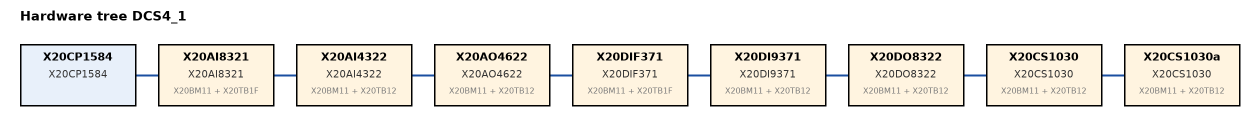
```
X20AI4322 : X20AI4322 v1.2.0.0  [SS1 -> X20TB12d.SS; SL -> X20BM11d.SL1]
X20AI8321 : X20AI8321 v1.5.0.0  [SS1 -> X20TB1F.SS; SL -> X20BM11a.SL1]
X20AO4622 : X20AO4622 v1.3.0.0  [SS1 -> X20TB12e.SS; SL -> X20BM11e.SL1]
  ChannelType01 = 4 to 20mA
  ChannelType02 = 4 to 20mA
  ChannelType03 = 4 to 20mA
  ChannelType04 = 4 to 20mA
X20BM11 : X20BM11 v1.1.0.0  [X2X1 -> X20BM11c.X2X2]
X20BM11a : X20BM11 v1.1.0.0  [X2X1 -> X20CP1584.IF6]
X20BM11b : X20BM11 v1.1.0.0  [X2X1 -> X20BM11e.X2X2]
X20BM11c : X20BM11 v1.1.0.0  [X2X1 -> X20BM11f.X2X2]
X20BM11d : X20BM11 v1.1.0.0  [X2X1 -> X20BM11a.X2X2]
X20BM11e : X20BM11 v1.1.0.0  [X2X1 -> X20BM11d.X2X2]
X20BM11f : X20BM11 v1.1.0.0  [X2X1 -> X20BM11b.X2X2]
X20BM11g : X20BM11 v1.1.0.0  [X2X1 -> X20BM11.X2X2]
X20CP1584 : X20CP1584 v1.10.0.0
  Connector IF2:
    ActivateDevice = 1
    Mode = Manual
    InternetAddress = 192.168.50.13
    SubnetMask = 255.255.255.0
  Connector IF3:
    DNAConfiguration = manual
  ConfigurationID = IP001_DCS2_2
  UserPartitionSize = 0
  Simulation = 1
  FileDevice1
  FileDeviceName1 = USER
  FileDevicePath1 = USER_PATH
  ActivateOpcUa = 1
  OpcUa_AuthenticationSecurityPolicy_EnableNone = 1
  OpcUa_AuthenticationSecurityPolicy_EnableBasic128Rsa15 = 1
  OpcUaInformationModels_PV_Version = 1
X20CS1030 : X20CS1030 v1.8.0.0  [SS1 -> X20TB12a.SS; SL -> X20BM11.SL1]
X20CS1030a : X20CS1030 v1.8.0.0  [SS1 -> X20TB12.SS; SL -> X20BM11g.SL1]
X20DI9371 : X20DI9371 v1.3.0.0  [SS1 -> X20TB12b.SS; SL -> X20BM11f.SL1]
X20DIF371 : X20DIF371 v1.2.0.0  [SS1 -> X20TB1F1.SS; SL -> X20BM11b.SL1]
X20DO8322 : X20DO8322 v1.4.0.0  [SS1 -> X20TB12c.SS; SL -> X20BM11c.SL1]
X20TB12 : X20TB12 v1.0.0.0
X20TB12a : X20TB12 v1.0.0.0
X20TB12b : X20TB12 v1.0.0.0
X20TB12c : X20TB12 v1.0.0.0
X20TB12d : X20TB12 v1.0.0.0
X20TB12e : X20TB12 v1.0.0.0
X20TB1F : X20TB1F v1.0.0.0
X20TB1F1 : X20TB1F v1.0.0.0
```

### IoMap.iom - X20CP1584/IoMap.iom
```iecst
VAR_CONFIG
	::DCS4_1:AI[1,1].RAW AT %IW."X20AI8321".AnalogInput01;
	::DCS4_1:AI[1,2].RAW AT %IW."X20AI8321".AnalogInput02;
	::DCS4_1:AI[1,3].RAW AT %IW."X20AI8321".AnalogInput03;
	::DCS4_1:AI[1,4].RAW AT %IW."X20AI8321".AnalogInput04;
	::DCS4_1:AI[1,5].RAW AT %IW."X20AI8321".AnalogInput05;
	::DCS4_1:AI[1,6].RAW AT %IW."X20AI8321".AnalogInput06;
	::DCS4_1:AI[1,7].RAW AT %IW."X20AI8321".AnalogInput07;
	::DCS4_1:AI[1,8].RAW AT %IW."X20AI8321".AnalogInput08;
	::DCS4_1:AI[2,1].RAW  AT %IW."X20AI4322".AnalogInput01;
	::DCS4_1:AI[2,2].RAW  AT %IW."X20AI4322".AnalogInput02;
	::DCS4_1:AI[2,3].RAW  AT %IW."X20AI4322".AnalogInput03;
	::DCS4_1:AI[2,4].RAW  AT %IW."X20AI4322".AnalogInput04;
	::DCS4_1:AO[1,1].RAW AT %QW."X20AO4622".AnalogOutput01;
	::DCS4_1:DI[1,1].In AT %IX."X20DIF371".DigitalInput01;
	::DCS4_1:DI[1,2].In AT %IX."X20DIF371".DigitalInput02;
	::DCS4_1:DI[1,3].In AT %IX."X20DIF371".DigitalInput03;
	::DCS4_1:DI[1,4].In AT %IX."X20DIF371".DigitalInput04;
	::DCS4_1:DO_[1,1].Out AT %QX."X20DO8322".DigitalOutput01;
	::DCS4_1:DO_[1,2].Out AT %QX."X20DO8322".DigitalOutput02;
	::DCS4_1:DO_[1,3].Out AT %QX."X20DO8322".DigitalOutput03;
	::DCS4_1:DO_[1,4].Out AT %QX."X20DO8322".DigitalOutput04;
	::DCS4_1:DO_[1,5].Out AT %QX."X20DO8322".DigitalOutput05;
	::DCS4_1:DO_[1,6].Out AT %QX."X20DO8322".DigitalOutput06;
	::DCS4_1:AO[1,2].RAW AT %QW."X20AO4622".AnalogOutput02;
	::DCS4_1:AO[1,3].RAW AT %QW."X20AO4622".AnalogOutput03;
	::DCS4_1:AO[1,4].RAW AT %QW."X20AO4622".AnalogOutput04;
	::DCS4_1:DI[1,5].In AT %IX."X20DIF371".DigitalInput05;
	::DCS4_1:DI[1,6].In AT %IX."X20DIF371".DigitalInput06;
	::DCS4_1:DI[1,7].In AT %IX."X20DIF371".DigitalInput07;
	::DCS4_1:DI[1,8].In AT %IX."X20DIF371".DigitalInput08;
	::DCS4_1:DI[1,9].In AT %IX."X20DIF371".DigitalInput09;
	::DCS4_1:DI[1,10].In AT %IX."X20DIF371".DigitalInput10;
	::DCS4_1:DI[1,11].In AT %IX."X20DIF371".DigitalInput11;
	::DCS4_1:DI[1,12].In AT %IX."X20DIF371".DigitalInput12;
	::DCS4_1:DI[1,13].In AT %IX."X20DIF371".DigitalInput13;
	::DCS4_1:DI[1,14].In AT %IX."X20DIF371".DigitalInput14;
	::DCS4_1:DI[1,15].In AT %IX."X20DIF371".DigitalInput15;
	::DCS4_1:DI[1,16].In AT %IX."X20DIF371".DigitalInput16;
	::DCS4_1:DI[2,1].In  AT %IX."X20DI9371".DigitalInput01;
	::DCS4_1:DI[2,2].In  AT %IX."X20DI9371".DigitalInput02;
	::DCS4_1:DI[2,3].In  AT %IX."X20DI9371".DigitalInput03;
	::DCS4_1:DI[2,4].In  AT %IX."X20DI9371".DigitalInput04;
	::DCS4_1:DI[2,5].In  AT %IX."X20DI9371".DigitalInput05;
	::DCS4_1:DI[2,6].In  AT %IX."X20DI9371".DigitalInput06;
	::DCS4_1:DI[2,7].In  AT %IX."X20DI9371".DigitalInput07;
	::DCS4_1:DI[2,8].In  AT %IX."X20DI9371".DigitalInput08;
	::DCS4_1:DI[2,9].In  AT %IX."X20DI9371".DigitalInput09;
	::DCS4_1:DI[2,10].In  AT %IX."X20DI9371".DigitalInput10;
	::DCS4_1:DI[2,11].In  AT %IX."X20DI9371".DigitalInput11;
	::DCS4_1:DI[2,12].In  AT %IX."X20DI9371".DigitalInput12;
	::DCS4_1:DO_[1,7].Out AT %QX."X20DO8322".DigitalOutput07;
	::DCS4_1:DO_[1,8].Out AT %QX."X20DO8322".DigitalOutput08;
END_VAR
```

## Configuration DCS5_1

CPU X20CP1584, AutomationRuntime B4.92, Build 4.1.2, Vc V4.72.5

### Hardware
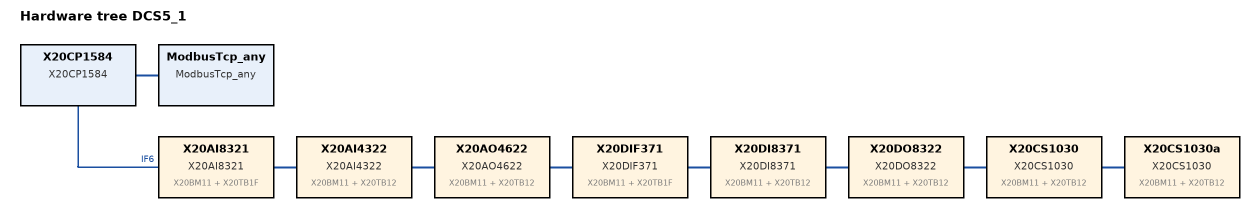
```
ModbusTcp_any : ModbusTcp_any v1.1.0.0  [ETH1 -> X20CP1584.IF2 [Cable Type=PowerlinkCable, Length=10, Version=1.0.0.3]]
  IpAddress = 192.168.50.114
  UnitId = 1
X20AI4322 : X20AI4322 v1.2.0.0  [SS1 -> X20TB12d.SS; SL -> X20BM11d.SL1]
  Supervision = off
X20AI8321 : X20AI8321 v1.5.0.0  [SS1 -> X20TB1F.SS; SL -> X20BM11a.SL1]
  Supervision = off
X20AO4622 : X20AO4622 v1.3.0.0  [SS1 -> X20TB12e.SS; SL -> X20BM11e.SL1]
  Supervision = off
  ChannelType01 = 4 to 20mA
  ChannelType02 = 4 to 20mA
  ChannelType03 = 4 to 20mA
  ChannelType04 = 4 to 20mA
X20BM11 : X20BM11 v1.1.0.0  [X2X1 -> X20BM11c.X2X2]
X20BM11a : X20BM11 v1.1.0.0  [X2X1 -> X20CP1584.IF6]
X20BM11b : X20BM11 v1.1.0.0  [X2X1 -> X20BM11e.X2X2]
X20BM11c : X20BM11 v1.1.0.0  [X2X1 -> X20BM11f.X2X2]
X20BM11d : X20BM11 v1.1.0.0  [X2X1 -> X20BM11a.X2X2]
X20BM11e : X20BM11 v1.1.0.0  [X2X1 -> X20BM11d.X2X2]
X20BM11f : X20BM11 v1.1.0.0  [X2X1 -> X20BM11b.X2X2]
X20BM11g : X20BM11 v1.1.0.0  [X2X1 -> X20BM11.X2X2]
X20CP1584 : X20CP1584 v1.10.0.0
  Connector IF2:
    ActivateDevice = 1
    Mode = Manual
    InternetAddress = 192.168.50.14
    SubnetMask = 255.255.255.0
    ActivateModbus = 1
    NumSlaves = -1
    NumAllBlocks = -1
    MemSizeIn = -1
    MemSizeOut = -1
  Connector IF3:
    DNAConfiguration = manual
  ConfigurationID = IP001_DCS2_2
  UserPartitionSize = 0
  Simulation = 1
  FileDevice1
  FileDeviceName1 = USER
  FileDevicePath1 = USER_PATH
  ActivateOpcUa = 1
  OpcUa_AuthenticationSecurityPolicy_EnableNone = 1
  OpcUa_AuthenticationSecurityPolicy_EnableBasic128Rsa15 = 1
  OpcUaInformationModels_PV_Version = 1
X20CS1030 : X20CS1030 v1.8.0.0  [SS1 -> X20TB12a.SS; SL -> X20BM11.SL1]
  Supervision = off
X20CS1030a : X20CS1030 v1.8.0.0  [SS1 -> X20TB12.SS; SL -> X20BM11g.SL1]
  Supervision = off
X20DI8371 : X20DI8371 v1.3.0.0  [SS1 -> X20TB12b.SS; SL -> X20BM11f.SL1]
  Supervision = off
X20DIF371 : X20DIF371 v1.2.0.0  [SS1 -> X20TB1F1.SS; SL -> X20BM11b.SL1]
  Supervision = off
X20DO8322 : X20DO8322 v1.4.0.0  [SS1 -> X20TB12c.SS; SL -> X20BM11c.SL1]
  Supervision = off
X20TB12 : X20TB12 v1.0.0.0
X20TB12a : X20TB12 v1.0.0.0
X20TB12b : X20TB12 v1.0.0.0
X20TB12c : X20TB12 v1.0.0.0
X20TB12d : X20TB12 v1.0.0.0
X20TB12e : X20TB12 v1.0.0.0
X20TB1F : X20TB1F v1.0.0.0
X20TB1F1 : X20TB1F v1.0.0.0
```

### IoMap.iom - X20CP1584/IoMap.iom
```iecst
VAR_CONFIG
	::DCS5_1:AI[1,1].RAW AT %IW."X20AI8321".AnalogInput01;
	::DCS5_1:AI[1,2].RAW AT %IW."X20AI8321".AnalogInput02;
	::DCS5_1:AI[1,3].RAW AT %IW."X20AI8321".AnalogInput03;
	::DCS5_1:AI[1,4].RAW AT %IW."X20AI8321".AnalogInput04;
	::DCS5_1:AI[1,5].RAW AT %IW."X20AI8321".AnalogInput05;
	::DCS5_1:AI[1,6].RAW AT %IW."X20AI8321".AnalogInput06;
	::DCS5_1:AI[1,7].RAW AT %IW."X20AI8321".AnalogInput07;
	::DCS5_1:AI[1,8].RAW AT %IW."X20AI8321".AnalogInput08;
	::DCS5_1:AI[2,1].RAW AT %IW."X20AI4322".AnalogInput01;
	::DCS5_1:AI[2,2].RAW AT %IW."X20AI4322".AnalogInput02;
	::DCS5_1:AI[2,3].RAW AT %IW."X20AI4322".AnalogInput03;
	::DCS5_1:AI[2,4].RAW AT %IW."X20AI4322".AnalogInput04;
	::DCS5_1:AO[1,1].RAW AT %QW."X20AO4622".AnalogOutput01;
	::DCS5_1:DI[1,1].In AT %IX."X20DIF371".DigitalInput01;
	::DCS5_1:DI[1,2].In AT %IX."X20DIF371".DigitalInput02;
	::DCS5_1:DI[1,3].In AT %IX."X20DIF371".DigitalInput03;
	::DCS5_1:DI[1,4].In AT %IX."X20DIF371".DigitalInput04;
	::DCS5_1:DO_[1,1].Out AT %QX."X20DO8322".DigitalOutput01;
	::DCS5_1:DO_[1,2].Out AT %QX."X20DO8322".DigitalOutput02;
	::DCS5_1:DO_[1,3].Out AT %QX."X20DO8322".DigitalOutput03;
	::DCS5_1:DO_[1,4].Out AT %QX."X20DO8322".DigitalOutput04;
	::DCS5_1:DO_[1,5].Out AT %QX."X20DO8322".DigitalOutput05;
	::DCS5_1:DO_[1,6].Out AT %QX."X20DO8322".DigitalOutput06;
	::DCS5_1:AO[1,2].RAW AT %QW."X20AO4622".AnalogOutput02;
	::DCS5_1:AO[1,3].RAW AT %QW."X20AO4622".AnalogOutput03;
	::DCS5_1:AO[1,4].RAW AT %QW."X20AO4622".AnalogOutput04;
	::DCS5_1:DI[1,5].In AT %IX."X20DIF371".DigitalInput05;
	::DCS5_1:DI[1,6].In AT %IX."X20DIF371".DigitalInput06;
	::DCS5_1:DI[1,7].In AT %IX."X20DIF371".DigitalInput07;
	::DCS5_1:DI[1,8].In AT %IX."X20DIF371".DigitalInput08;
	::DCS5_1:DI[1,9].In AT %IX."X20DIF371".DigitalInput09;
	::DCS5_1:DI[1,10].In AT %IX."X20DIF371".DigitalInput10;
	::DCS5_1:DI[1,11].In AT %IX."X20DIF371".DigitalInput11;
	::DCS5_1:DI[1,12].In AT %IX."X20DIF371".DigitalInput12;
	::DCS5_1:DI[1,13].In AT %IX."X20DIF371".DigitalInput13;
	::DCS5_1:DI[1,14].In AT %IX."X20DIF371".DigitalInput14;
	::DCS5_1:DI[1,15].In AT %IX."X20DIF371".DigitalInput15;
	::DCS5_1:DI[1,16].In AT %IX."X20DIF371".DigitalInput16;
	::DCS5_1:DI[2,1].In AT %IX."X20DI8371".DigitalInput01;
	::DCS5_1:DI[2,2].In AT %IX."X20DI8371".DigitalInput02;
	::DCS5_1:DI[2,3].In AT %IX."X20DI8371".DigitalInput03;
	::DCS5_1:DI[2,4].In AT %IX."X20DI8371".DigitalInput04;
	::DCS5_1:DI[2,5].In AT %IX."X20DI8371".DigitalInput05;
	::DCS5_1:DI[2,6].In AT %IX."X20DI8371".DigitalInput06;
	::DCS5_1:DI[2,7].In AT %IX."X20DI8371".DigitalInput07;
	::DCS5_1:DI[2,8].In AT %IX."X20DI8371".DigitalInput08;
	::DCS5_1:DO_[1,7].Out AT %QX."X20DO8322".DigitalOutput07;
	::DCS5_1:DO_[1,8].Out AT %QX."X20DO8322".DigitalOutput08;
END_VAR
```

## Configuration DCS9_1

### Task classes (Cpu.sw)
```
Cyclic#4:
  DCS9_1 <- DCS9_1.prg
Libraries: Lib489, standard, AsMbTCP, AsBrStr, asstring, MTBasics, DRV_mbus, DataObj, operator, astime, AsIecCon, LibIP001, sys_lib, brsystem, MTTypes, dvframe, runtime
```

### Hardware
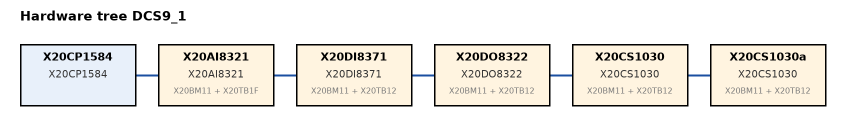
```
X20AI8321 : X20AI8321 v1.4.0.0  [SS1 -> X20TB1F.SS; SL -> X20BM11a.SL1]
  Supervision = off
X20BM11 : X20BM11 v1.0.0.1  [X2X1 -> X20BM11c.X2X2]
X20BM11a : X20BM11 v1.0.0.1  [X2X1 -> X20CP1584.IF6]
X20BM11b : X20BM11 v1.0.0.1  [X2X1 -> X20BM11a.X2X2]
X20BM11c : X20BM11 v1.0.0.1  [X2X1 -> X20BM11b.X2X2]
X20BM11d : X20BM11 v1.0.0.1  [X2X1 -> X20BM11.X2X2]
X20CP1584 : X20CP1584 v1.8.0.0
  Connector IF2:
    ActivateDevice = 1
    Mode = Manual
    InternetAddress = 192.168.50.15
    SubnetMask = 255.255.255.0
  ConfigurationID = IP001_DCS2_2
  ActivateOpcUa = 1
  OpcUa_AuthenticationSecurityPolicy_EnableNone = 1
  OpcUa_AuthenticationSecurityPolicy_EnableBasic128Rsa15 = 1
  OpcUaInformationModels_PV_Version = 1
X20CS1030 : X20CS1030 v1.7.0.0  [SS1 -> X20TB12.SS; SL -> X20BM11.SL1]
  Supervision = off
X20CS1030a : X20CS1030 v1.7.0.0  [SS1 -> X20TB12a.SS; SL -> X20BM11d.SL1]
  Supervision = off
X20DI8371 : X20DI8371 v1.0.2.0  [SS1 -> X20TB12b.SS; SL -> X20BM11b.SL1]
  Supervision = off
X20DO8322 : X20DO8322 v1.1.0.0  [SS1 -> X20TB12c.SS; SL -> X20BM11c.SL1]
  Supervision = off
X20TB12 : X20TB12 v1.0.0.0
X20TB12a : X20TB12 v1.0.0.0
X20TB12b : X20TB12 v1.0.0.0
X20TB12c : X20TB12 v1.0.0.0
X20TB1F : X20TB1F v1.0.0.0
```

### IoMap.iom - X20CP1584/IoMap.iom
```iecst
VAR_CONFIG
	::DCS9_1:DI[1,1].In AT %IX."X20DI8371".DigitalInput01;
	::DCS9_1:DI[1,2].In AT %IX."X20DI8371".DigitalInput02;
	::DCS9_1:DI[1,3].In AT %IX."X20DI8371".DigitalInput03;
	::DCS9_1:DI[1,4].In AT %IX."X20DI8371".DigitalInput04;
	::DCS9_1:AI[1,1].RAW AT %IW."X20AI8321".AnalogInput01;
	::DCS9_1:AI[1,2].RAW AT %IW."X20AI8321".AnalogInput02;
	::DCS9_1:AI[1,3].RAW AT %IW."X20AI8321".AnalogInput03;
	::DCS9_1:AI[1,4].RAW AT %IW."X20AI8321".AnalogInput04;
	::DCS9_1:AI[1,5].RAW AT %IW."X20AI8321".AnalogInput05;
	::DCS9_1:AI[1,6].RAW AT %IW."X20AI8321".AnalogInput06;
	::DCS9_1:AI[1,7].RAW AT %IW."X20AI8321".AnalogInput07;
	::DCS9_1:AI[1,8].RAW AT %IW."X20AI8321".AnalogInput08;
	::DCS9_1:DO_[1,1].Out AT %QX."X20DO8322".DigitalOutput01;
	::DCS9_1:DO_[1,2].Out AT %QX."X20DO8322".DigitalOutput02;
	::DCS9_1:DO_[1,3].Out AT %QX."X20DO8322".DigitalOutput03;
	::DCS9_1:DO_[1,4].Out AT %QX."X20DO8322".DigitalOutput04;
	::DCS9_1:DO_[1,5].Out AT %QX."X20DO8322".DigitalOutput05;
	::DCS9_1:DO_[1,6].Out AT %QX."X20DO8322".DigitalOutput06;
	::DCS9_1:DI[1,5].In AT %IX."X20DI8371".DigitalInput05;
	::DCS9_1:DI[1,6].In AT %IX."X20DI8371".DigitalInput06;
	::DCS9_1:DI[1,7].In AT %IX."X20DI8371".DigitalInput07;
	::DCS9_1:DI[1,8].In AT %IX."X20DI8371".DigitalInput08;
	::DCS9_1:DO_[1,7].Out  AT %QX."X20DO8322".DigitalOutput07;
	::DCS9_1:DO_[1,8].Out AT %QX."X20DO8322".DigitalOutput08;
END_VAR
```

## Configuration stend

CPU X20CP3586, AutomationRuntime B4.92, Build 4.1.2, Vc V4.72.5

### Task classes (Cpu.sw)
```
Cyclic#1:
  str_test <- (binary)
Cyclic#4:
  DCS2_2 <- DCS2_2.prg
  DCS4_1 <- DCS4_1.prg
  DCS5_1 <- DCS5_1.prg
  DCS9_1 <- DCS9_1.prg
  DCS13_1 <- DCS13_1.prg
  DCS15_1 <- DCS15_1.prg
  DCS18_1 <- DCS18_1.prg
  DCS31_1 <- DCS31_1.prg
  DCS31_2 <- DCS31_2.prg
  DCS31_3 <- DCS31_3.prg
  DCS31_4 <- DCS31_4.prg
  DCS34_1 <- DCS34_1.prg
  DCS35_1 <- DCS35_1.prg
  DCS36_1 <- DCS36_1.prg
  DCS37_1 <- DCS37_1.prg
  DCS39_1 <- DCS39_1.prg
  DCS40_1 <- DCS40_1.prg
  DCS45_1 <- DCS45_1.prg
Binaries: udbdef, TCData, arconfig, User, Role, iomap, asfw, ashwac, ashwd, sysconf, asrrad, OpcUaMap
Libraries: operator, astime, AsIecCon, Lib489, LibIP001, AsBrStr, DRV_mbus, DataObj, dvframe, runtime, MTBasics, brsystem, MTTypes, sys_lib, standard, AsMbTCP, asstring, asarcfg
```

### Hardware
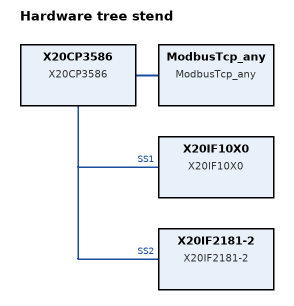
```
ModbusTcp_any : ModbusTcp_any v1.1.0.0  [ETH1 -> X20CP3586.IF2 [Cable Type=PowerlinkCable, Length=10, Version=1.0.0.3]]
  IpAddress = 192.168.15.202
  UnitId = 1
X20CP3586 : X20CP3586 v1.10.0.0
  Connector IF2:
    ActivateDevice = 1
    EthInterfaceRedundant = 1
    ClusterInternetAddress = 192.168.15.210
    ClusterSubnetMask = 255.255.255.0
    Mode = FromCluster
    PrimaryHostName = pri-br-automation
    PrimaryInternetAddress = 192.168.15.211
    SecondaryHostName = sec-br-automation
    SecondaryInternetAddress = 192.168.15.212
    RedundantInaSelector = RedundantIna
    InaCluster = 1
    InaCNodeNumber = 10
    ActivateModbus = 1
    NumSlaves = -1
    NumAllBlocks = -1
    MemSizeIn = -1
    MemSizeOut = -1
  Connector IF3:
    Operation = EthOnly
    EplEthInterfaceRedundant = 1
    EthernetMode = DHCP Client
    PrimaryHostName = pri-br-automation
    SecondaryHostName = sec-br-automation
    RedundantInaSelector = RedundantIna
  ConfigurationID = OI551_X20CP3584
  UserPartitionSize = 0
  RemanentGlobalPvSize = 15000
  TimerDeviceType = RIF
  Cyclic8Duration = 100000
  FileDevice1
  FileDeviceName1 = USER
  FileDevicePath1 = USER_PATH
  ActivateSntpServer = 1
  ActivateSntp = 1
  SntpcServAddr1 = 192.168.15.58
  SntpcServAddr2 = 192.168.15.58
  SntpcServAddr3 = 192.168.15.58
  SntpcServAddr4 = 192.168.15.58
  EthernetDefaultGateway = 192.168.15.254
  ActivateOpcUa = 1
  OpcUa_AuthenticationSecurityPolicy_EnableNone = 1
  OpcUa_AuthenticationSecurityPolicy_EnableBasic128Rsa15 = 1
  OpcUa_Limits_MaxReferencesToReturn = 100000
  OpcUa_Limits_MonitoredItemsPerSubscription = 100000
  OpcUaMaxSubsItemQueueSize = 1000
  OpcUaInformationModels_PV_Version = 2
  ActivateRedundancy = 1
X20IF10X0 : X20IF10X0 v1.3.0.0  [IF1 -> X20IF10X0 - redundant.IF1 (TargetRedundancyModule=True); SS -> X20CP3586.SS1]
X20IF2181-2 : X20IF2181-2 v1.9.0.0  [SS -> X20CP3586.SS2]
  Connector IF1:
    DNAConfiguration = manual
    EplInterfaceRedundant = 1
    Mode = RMN
    EplEthInterfaceRedundant = 1
    EthernetMode = Manual
    RedundantInaSelector = RedundantIna
```

## Logical view

Binary libraries used (declarations not repeated): operator, runtime, astime, AsIecCon, standard, AsMbTCP, AsBrStr, asstring, MTBasics 5.06.0, DRV_mbus, DataObj, sys_lib, brsystem, MTTypes 1.03.4, dvframe

### Package Logical/Libraries - Global libraries

### Library Logical/Libraries/Lib489 (IEC) - Lib ASUTP
Depends on: MTBasics, standard, AsMbTCP, asstring, DRV_mbus, AsBrStr

#### Types.typ - Exported data types
```iecst
TYPE
	tUVP_Data : 	STRUCT
		Time : tTime;
		LineCurrent : ARRAY[1..16]OF tUVP_Line_Current;
		Prev_hour : ARRAY[1..16]OF tUVP_prev_hour;
		Prev_day : ARRAY[1..16]OF tUVP_prev_day;
		NTP : tNTP;
		MR_113 : tMR113_03;
		MR_113_new : tMR113_03;
		Byte_order : UINT;
		Byte_order_new : UINT := 8961; (*16#2301*)
		synchrooo : BOOL;
		DeltaTime : INT;
		read_gas_comp : BOOL;
		write_gas_comp : BOOL;
	END_STRUCT;
	tTime : 	STRUCT
		Day : UINT;
		Month : UINT;
		Year : UINT;
		Hour : UINT;
		Min : UINT;
		Sec : UINT;
		TPs : UINT;
	END_STRUCT;
	tUVP_Line_Current : 	STRUCT  (*Тип текущих параметров измерительного трубопровода*)
		Pressure : REAL; (*Избыточное давление, Па*)
		Pressure_absolut : REAL; (*Абсолютное давление, Па*)
		Temperature : REAL; (*Температура, С*)
		Enthalpy : REAL; (*Энтальпия, Дж/кг*)
		Mass_flow : REAL; (*Массовый расход, кг/с*)
		Massa : REAL; (*Масса (накопительный параметр), кг*)
		Volume_r_u : REAL; (*Объем в рабочих условиях (накопительный параметр), м3*)
		Volume_st_u : REAL; (*Объем в стандартных условиях (накопительный параметр), м3*)
		Heat_power : REAL; (*Тепловая мощность, Вт*)
		Heat_energy : REAL; (*Тепловая энергия	(накопительный параметр), Дж*)
		Time_staff_work : UDINT; (*Время штатной работы (накопительный параметр), сек*)
		Time_supernumerary_situations : UDINT; (*Время нештатных ситуаций (накопительный параметр), сек*)
		Parameter_sensor_mass_flow : REAL; (*Параметр датчика расхода/количества (массовый расход), кг/с*)
		Parameter_sensor_vol_flow_r_u : REAL; (*Параметр датчика расхода/количества (объемный расход в р.у.), м3/с*)
		Parameter_sensor_vol_flow_st_u : REAL; (*Параметр датчика расхода/количества (объемный расход в ст.у.), м3/с*)
		Parameter_sensor_massa : REAL; (*Параметр датчика расхода/количества (масса) (накопительный параметр), кг*)
		Parameter_sensor_volume : REAL; (*Параметр датчика расхода/количества (объемный расход в р.у.) (накопительный параметр), м3*)
		Quantity_errors : UINT; (*Количество ошибок на трубопроводе*)
		Level_errors : UINT; (*Уровень критичности ошибок трубопровода*)
		Density_st_u : REAL; (*Плотность среды в стандартных условиях, кг/м3*)
		Density_r_u : REAL; (*Плотность измеряемой среды в рабочих условиях, кг/м3*)
		Difference_pressure_SU : REAL; (*Перепад давления для трубопроводов на СУ, Па*)
		Volume_flow_st_u : REAL; (*Объемный расход в ст.у., м3/с*)
		Volume_flow_r_u : REAL; (*Объемный расход в р.у., м3/с*)
	END_STRUCT;
	tNTP : 	STRUCT
		IPAddr1 : UINT;
		IPAddr2 : UINT;
		cmd : UINT;
		IpAddress1 : USINT;
		IpAddress2 : USINT;
		IpAddress3 : USINT;
		IpAddress4 : USINT;
	END_STRUCT;
	tMR113_03 : 	STRUCT  (*Тип управления параметрами среды*)
		MolarMass : UINT; (*Молярная/массовая концентрация*)
		AbsRelate : UINT; (*Влажность задается абсолютным/относительным значением*)
		CH4 : REAL;
		C2H6 : REAL;
		C3H8 : REAL;
		nC4H10 : REAL;
		iC4H10 : REAL;
		nC5H12 : REAL;
		N2 : REAL;
		CO2 : REAL;
		H2O : REAL;
		H2S : REAL;
		C6H14 : REAL;
		C7H16 : REAL;
		O2 : REAL;
		iC5H12 : REAL;
		AbsH2O : REAL;
	END_STRUCT;
	tUVP_prev_hour : 	STRUCT  (*Тип количественных показателей за предыдущий час/2 часа*)
		Massa : REAL; (*Масса, кг*)
		Volume_r_u : REAL; (*Объем в рабочих условиях, м3*)
		Volume_st_u : REAL; (*Объем в стандартных условиях, м3*)
		Parameter_sensor_massa : REAL; (*Параметр датчика расхода/количества (масса), кг*)
		Parameter_sensor_volume_r_u : REAL; (*Параметр датчика расхода/количества (объем в р.у.), м3*)
	END_STRUCT;
	tUVP_prev_day : 	STRUCT  (*Тип количественных показателей за предыдущие сутки*)
		Massa : REAL; (*Масса, кг*)
		Volume_r_u : REAL; (*Объем в рабочих условиях, м3*)
		Volume_st_u : REAL; (*Объем в стандартных условиях, м3*)
		Parameter_sensor_massa : REAL; (*Параметр датчика расхода/количества (масса), кг*)
		Parameter_sensor_volume_r_u : REAL; (*Параметр датчика расхода/количества (объем в р.у.), м3*)
	END_STRUCT;
	tAuma_write : 	STRUCT
		cmd : UINT;
		Pos : UINT;
	END_STRUCT;
	tAuma_read : 	STRUCT
		state_1 : UINT;
		state_2 : UINT;
		Pos : UINT;
	END_STRUCT;
END_TYPE
```

#### Lib489.fun - Exported functions and function blocks
```iecst
{REDUND_OK} FUNCTION_BLOCK UVP_TCP (*UVP_MB_TCP*) (*$GROUP=User,$CAT=User,$GROUPICON=User.png,$CATICON=User.png*)
	VAR_INPUT
		pPort : UDINT;
	END_VAR
	VAR
		status : UINT;
		state : UINT;
		step : USINT;
		req_3x : mbReadHoldingRegisters;
		req_4x : mbReadInputRegisters;
		req_6x : mbWriteSingleRegister;
		req_16x : mbWriteMultipleRegisters;
		UVP_Data : tUVP_Data := (NTP:=(cmd:=13579,IpAddress1:=192,IpAddress2:=168,IpAddress3:=50,IpAddress4:=12));
		curTP : USINT;
		Timeout_T : TON;
	END_VAR
END_FUNCTION_BLOCK

{REDUND_OK} FUNCTION_BLOCK ABAK_TCP (*ABAK_MB_TCP*) (*$GROUP=User,$CAT=User,$GROUPICON=User.png,$CATICON=User.png*)
	VAR_INPUT
		pPort : BOOL;
	END_VAR
	VAR
		status : UINT;
		state : UINT;
		step : USINT;
		req_3x : mbReadHoldingRegisters;
		req_4x : mbReadInputRegisters;
		req_6x : mbWriteSingleRegister;
		req_16x : mbWriteMultipleRegisters;
		Timeout_T : TON;
	END_VAR
END_FUNCTION_BLOCK

{REDUND_OK} FUNCTION_BLOCK PassportValve (*ФБ для отображения ЗД по индексу*) (*$GROUP=User,$CAT=User,$GROUPICON=User.png,$CATICON=User.png*)
	VAR_INPUT
		index : {REDUND_UNREPLICABLE} USINT;
		is_first : BOOL;
	END_VAR
	VAR_IN_OUT
		Gate_buf : FValve;
	END_VAR
	VAR
		cmdOpen : BOOL;
		cmdClose : BOOL;
		cmdBlck : BOOL;
		cmdAuto : BOOL;
		cmdImit : BOOL;
		cmdResetAlarms : BOOL;
		statePLC_control : BOOL;
		stateLeak : BOOL;
		stateAuto : BOOL;
		stateManu : BOOL;
		stateOpening : BOOL;
		stateClosing : BOOL;
		stateOpened : BOOL;
		stateClosed : BOOL;
		statePAZ : BOOL;
		failTimeout : BOOL;
		failTimeoutO : BOOL;
		failTimeoutC : BOOL;
		timePT : DINT;
	END_VAR
END_FUNCTION_BLOCK

{REDUND_OK} FUNCTION_BLOCK PassportAI (*ФБ для отображения аналогового входа по индексу*) (*$GROUP=User,$CAT=User,$GROUPICON=User.png,$CATICON=User.png*)
	VAR_INPUT
		index1_old : USINT;
		index1 : USINT;
		index2_old : USINT;
		index2 : USINT;
		is_first : BOOL;
	END_VAR
	VAR_IN_OUT
		AI_buf : FAI;
	END_VAR
	VAR
		cmdImit : BOOL;
		cmdHiEn : BOOL;
		cmdHiHiEn : BOOL;
		cmdLoEn : BOOL;
		cmdLoLoEn : BOOL;
		stateInvalid : BOOL;
		stateHi : BOOL;
		stateHiHi : BOOL;
		stateLo : BOOL;
		stateLoLo : BOOL;
		LoScale : REAL;
		HiScale : REAL;
		HiLimit : REAL;
		HiHiLimit : REAL;
		LoLimit : REAL;
		LoLoLimit : REAL;
		current : REAL;
		Value : REAL;
		ImitVal : REAL;
	END_VAR
END_FUNCTION_BLOCK

{REDUND_OK} FUNCTION_BLOCK FValve (*Задвижка*) (*$GROUP=User,$CAT=User,$GROUPICON=User.png,$CATICON=User.png*)
	VAR_INPUT RETAIN
		r0 : UINT; (*Командное слово(бит0-Открыть,бит1-Закрыть,,бит2-Стоп,бит13-имитация,бит14-Сброс аварий)*)
	END_VAR
	VAR_INPUT
		AlarmDI : BOOL;
		OpenedDI : BOOL; (*DI Открыто*)
		ClosedDI : BOOL; (*DI Закрыто*)
		PAZ : BOOL; (*Кран под управлением ПАЗ*)
	END_VAR
	VAR_INPUT RETAIN
		FullTimerInterval : DINT := 30000; (*Время полного хода (мс)*)
	END_VAR
	VAR_OUTPUT
		CloseDO : BOOL; (*DO Закрыть*)
		OpenDO : BOOL; (*DO Открыть*)
		StopDO : BOOL; (*DO Стоп*)
		r1 : UINT; (*Состояние(бит1-Таймаут,бит4-Открывается,бит5-Закрывается,бит6-Открыт,бит7-Закрыт,бит10-Авария,бит11-Нет связи по RS)*)
		Failures : UINT; (*Аварии*)
		Auto : BOOL;
		Opened : BOOL; (*Состояние ОТКРЫТО*)
		Closed : BOOL; (*Состояние ЗАКРЫТО*)
	END_VAR
	VAR RETAIN
		OpenDIOld : BOOL;
		CloseDIOld : BOOL;
	END_VAR
	VAR
		OpenNoAllow : BOOL;
		CloseNoAllow : BOOL;
		NoOpenNoAllow : BOOL;
		NoCloseNoAllow : BOOL;
		StopPresent : BOOL; (*если 1 то сигналы DO длятся до конца или до стопа, иначе 1 сек*)
		Open : BOOL; (*Команда ОТКРЫТЬ*)
		Close : BOOL; (*Команда ЗАКРЫТЬ*)
		Stop : BOOL; (*Команда СТОП*)
		Block : BOOL; (*Блокировка от ПАЗ*)
		TimeoutC : BOOL; (*Не закрылась*)
		TimeoutO : BOOL; (*Не открылась*)
		Opening : BOOL; (*Открывается*)
		Closing : BOOL; (*Закрывается*)
	END_VAR
	VAR RETAIN
		Imitation : BOOL; (*Иммитация*)
		T : TON := (PT:=T#3s); (*Таймер хода*)
		TSignal : TON := (PT:=T#1s); (*Таймер DO сигналов (1сек)*)
	END_VAR
END_FUNCTION_BLOCK

{REDUND_OK} FUNCTION_BLOCK FPostGassing (*TODO: Add your comment here*) (*$GROUP=User,$CAT=User,$GROUPICON=User.png,$CATICON=User.png*)
	VAR_INPUT
		StatusAI : UINT; (*регистр r1 AI загазованности*)
		HS01 : BOOL; (*Кнопка опробывания сигнализации о загазованности*)
		HS02 : BOOL; (*Кнопка снятия звуковой сигнализации о загазованности*)
	END_VAR
	VAR_OUTPUT
		HL01 : BOOL; (*Сигнализация загазованности "ГАЗ 10%"*)
		HL02 : BOOL; (*Сигнализация загазованности "ГАЗ 20%"*)
		HA01 : BOOL; (*Оповещатель звуковой загазованности*)
		Level1 : BOOL; (*Первый уровень загазованности*)
		Level1_10min : BOOL;
		Level2 : BOOL; (*Второй уровень загазованности*)
	END_VAR
	VAR
		HS01_Old : BOOL; (*HS01 в предыущем цикле*)
		Level1Old : BOOL; (*Level1 в предыущем цикле*)
		Level2Old : BOOL; (*Level2 в предыущем цикле*)
		Sound : BOOL; (*Звуковая зигнализация*)
		T : TON;
	END_VAR
END_FUNCTION_BLOCK

{REDUND_OK} FUNCTION_BLOCK FPIDreg_r (*PID*) (*$GROUP=User,$CAT=User,$GROUPICON=User.png,$CATICON=User.png*)
	VAR_INPUT RETAIN
		enable : BOOL := TRUE; (*start*)
		invert : BOOL := TRUE;
		mode : USINT := 1; (*ПИД: 0-выкл, 1-авто, 2-ручной, 3-ручной на макс, 4-ручной на мин*)
	END_VAR
	VAR_INPUT
		state : USINT; (*Исполнитель: бит0-закрыт,бит1-открыт,бит2-местный,бит3-неисправность*)
	END_VAR
	VAR_INPUT RETAIN
		X_set : REAL; (*setvalue - уставка*)
	END_VAR
	VAR_INPUT
		X : REAL; (*actvalue - входное значение*)
		Y : REAL; (*текущее положение регулятора*)
	END_VAR
	VAR_INPUT RETAIN
		Y_min : REAL := 0; (*минимальное открытие регулятора*)
		Y_max : REAL := 100; (*максимальное открытие регулятора*)
		Y_man : REAL := 0; (*вых велчина при ручном управлении*)
		Gain : REAL := 0.27; (*P*)
		IntegrationTime : REAL := 0.62; (*I*)
		DerivativeTime : REAL := 0.16; (*D*)
		FilterTime : REAL := 0.6;
	END_VAR
	VAR_INPUT
		AlOpen : BOOL;
		AlClose : BOOL;
	END_VAR
	VAR_OUTPUT
		status : DINT; (*код ошибки пид регулятора*)
		Y_out : REAL; (*выходное значение*)
	END_VAR
	VAR
		MTBasicsPID_0 : MTBasicsPID;
	END_VAR
END_FUNCTION_BLOCK

{REDUND_OK} FUNCTION_BLOCK FMotor (*Пускатель*) (*$GROUP=User,$CAT=User,$GROUPICON=User.png,$CATICON=User.png*)
	VAR_INPUT
		Start : BOOL; (*Коанда: пуск*)
		Stop : BOOL; (*Команда: стоп*)
		RunDI : BOOL; (*Входной дискрет "Запущен"*)
		Reset : BOOL; (*Сброс*)
	END_VAR
	VAR_INPUT RETAIN
		Block : BOOL; (*Блокировка*)
		Imitation : BOOL; (*Имитация*)
	END_VAR
	VAR_INPUT
		ResetMH : BOOL; (*Сброс моточасов*)
	END_VAR
	VAR_OUTPUT
		StartDO : BOOL; (*Управление дискретом "Пуск"*)
		StopDO : BOOL; (*Управление дискретом "Стоп"*)
		Status : UINT;
		Started_old : BOOL;
		Started : BOOL; (*Запущен*)
		Stopped_old : BOOL;
		Stopped : BOOL; (*Остановлен*)
		MotoHours : REAL;
	END_VAR
	VAR
		Timeout : BOOL;
		MH : FMHCounter;
		T : TON;
	END_VAR
END_FUNCTION_BLOCK

{REDUND_OK} FUNCTION_BLOCK FMHCounter (*FMHCounter*) (*$GROUP=User,$CAT=User,$GROUPICON=User.png,$CATICON=User.png*)
	VAR_INPUT
		Run : BOOL;
		Reset : BOOL;
	END_VAR
	VAR_OUTPUT RETAIN
		Counter : REAL;
	END_VAR
	VAR RETAIN
		Tik : UINT := 6;
	END_VAR
	VAR
		T : TON;
	END_VAR
END_FUNCTION_BLOCK

{REDUND_OK} FUNCTION_BLOCK FDO (*DO*) (*$GROUP=User,$CAT=User,$GROUPICON=User.png,$CATICON=User.png*)
	VAR_INPUT
		In : BOOL; (*Входное из алгоритма*)
	END_VAR
	VAR_INPUT RETAIN
		Inv : BOOL; (*Инверсия*)
		Mask : BOOL; (*Имитированное значение*)
		MaskEn : BOOL; (*Включени имитации*)
	END_VAR
	VAR_OUTPUT
		Out : BOOL; (*Выходное значение на модуль*)
	END_VAR
END_FUNCTION_BLOCK

{REDUND_OK} FUNCTION_BLOCK FDISKRreg_r (*Дискретный регулятор*) (*$GROUP=User,$CAT=User,$GROUPICON=User.png,$CATICON=User.png*)
	VAR_INPUT
		enable : BOOL;
	END_VAR
	VAR_INPUT RETAIN
		invert : BOOL;
		X_set_low : REAL;
		X_set_high : REAL;
	END_VAR
	VAR_INPUT
		X : REAL;
	END_VAR
	VAR_OUTPUT
		OnDO : BOOL;
		OffDO : BOOL;
	END_VAR
END_FUNCTION_BLOCK

{REDUND_OK} FUNCTION_BLOCK FDI (*DI*) (*$GROUP=User,$CAT=User,$GROUPICON=User.png,$CATICON=User.png*)
	VAR_INPUT
		In : BOOL; (*Входное значнеи с модуля*)
	END_VAR
	VAR_INPUT RETAIN
		Inv : BOOL; (*Инверсия*)
		Mask : BOOL; (*Имитированное значение*)
		MaskEn : BOOL; (*Включение имитации*)
	END_VAR
	VAR_OUTPUT
		Out : BOOL; (*Результирующее значение*)
	END_VAR
END_FUNCTION_BLOCK

{REDUND_OK} FUNCTION_BLOCK FAO (*AO*) (*$GROUP=User,$CAT=User,$GROUPICON=User.png,$CATICON=User.png*)
	VAR_INPUT
		HiHiEnabled : BOOL; (*Включение верхней аварии*)
		HiEnabled : BOOL; (*Включение верхнего предупреждения*)
		LoEnabled : BOOL; (*Включение нижнего предупреждения*)
		LoLoEnabled : BOOL; (*Включение нижней аварии*)
	END_VAR
	VAR_INPUT RETAIN
		HiHiLimit : REAL; (*Верхний аварийный предел*)
		HiLimit : REAL; (*Верхний технологический предел*)
		LoLimit : REAL; (*Нижний технологический предел*)
		LoLoLimit : REAL; (*Нижний аварийный предел*)
		Replace_Value : REAL; (*Подстановочное значение*)
		ImitationEn : BOOL; (*Включение имитации*)
	END_VAR
	VAR_INPUT
		CurrentOK : BOOL := TRUE; (*Ток в норме (для ПАЗ)*)
		CannelOK : BOOL := TRUE; (*Канал в норме (для ПАЗ)*)
	END_VAR
	VAR_INPUT RETAIN
		r0 : UINT; (*Регистр команд*)
	END_VAR
	VAR_INPUT
		Diff : BOOL := FALSE; (*Признак дифф. канала*)
		Safe : BOOL := FALSE; (*TRUE для ПАЗ*)
	END_VAR
	VAR_INPUT RETAIN
		LoScale : REAL; (*Нижний предел измерения*)
		HiScale : REAL; (*Верхний предел измерения*)
	END_VAR
	VAR_INPUT
		Value : REAL; (*Параметр в инженерных единицах*)
	END_VAR
	VAR_OUTPUT
		RAW : INT; (*Код АЦП*)
		RAW1 : INT; (*Код 2-го АЦП (для ПАЗ)*)
		HiHiAlarm : BOOL; (*Верхняя авария*)
		HiAlarm : BOOL; (*Верхнее предупреждение*)
		LoAlarm : BOOL; (*Нижнее предупреждение*)
		LoLoAlarm : BOOL; (*Нижняя авария*)
		Current : REAL; (*Ток (4-20 мА)*)
		Invalid : BOOL; (*Недостоверный сигнал*)
		r1 : UINT; (*Регистр состояний*)
		HiHiLimitPAZ : INT;
	END_VAR
	VAR
		Scale : REAL; (*Шкала датчика*)
	END_VAR
END_FUNCTION_BLOCK

{REDUND_OK} FUNCTION_BLOCK FAI (*AI*) (*$GROUP=User,$CAT=User,$GROUPICON=User.png,$CATICON=User.png*)
	VAR_INPUT
		RAW : INT; (*Код АЦП*)
	END_VAR
	VAR_INPUT RETAIN
		ChannelType : USINT; (*Тип канала(0-0-20мА,1-4-20мА,2-0-22мА,3-MB)*)
	END_VAR
	VAR_INPUT
		ChannelUnderflow : BOOL; (*Статус канала(обрыв)*)
		ChannelOverflow : BOOL; (*Статус канала(КЗ)*)
	END_VAR
	VAR_INPUT RETAIN
		HiScale : REAL; (*Верхний предел измерения*)
		LoScale : REAL; (*Нижний предел измерения*)
		ImitationEn : BOOL; (*Включение имитации*)
	END_VAR
	VAR_INPUT
		HiHiEnabled : BOOL; (*Включение верхней аварии*)
		HiEnabled : BOOL; (*Включение верхнего предупреждения*)
		LoEnabled : BOOL; (*Включение нижнего предупреждения*)
		LoLoEnabled : BOOL; (*Включение нижней аварии*)
	END_VAR
	VAR_INPUT RETAIN
		HiHiLimit : REAL; (*Верхний аварийный предел*)
		HiLimit : REAL; (*Верхний технологический предел*)
		LoLimit : REAL; (*Нижний технологический предел*)
		LoLoLimit : REAL; (*Нижний аварийный предел*)
		Replace_Value : REAL; (*Подстановочное значение*)
	END_VAR
	VAR_INPUT
		Hyst : REAL; (*Гистерезис*)
	END_VAR
	VAR_INPUT RETAIN
		RegCmd : USINT;
	END_VAR
	VAR_INPUT
		MbValue : REAL; (*Значение с Модбас*)
	END_VAR
	VAR_OUTPUT
		Invalid : BOOL; (*Недостоверный сигнал*)
		HiHiAlarm : BOOL; (*Верхняя авария*)
		HiAlarm : BOOL; (*Верхнее предупреждение*)
		LoAlarm : BOOL; (*Нижнее предупреждение*)
		LoLoAlarm : BOOL; (*Нижняя авария*)
		Value : REAL; (*Параметр в инженерных единицах*)
		Current : REAL; (*Ток (4-20 мА)*)
		Color : USINT; (*Цвет*)
		RegStatus : USINT;
	END_VAR
	VAR
		Scale : REAL; (*Шкала датчика*)
	END_VAR
END_FUNCTION_BLOCK

{REDUND_OK} FUNCTION_BLOCK FTorch (*Torch*) (*$GROUP=User,$CAT=User,$GROUPICON=User.png,$CATICON=User.png*)
	VAR_INPUT
		Mode_Manual : {REDUND_UNREPLICABLE} BOOL;
		Di_Fire : {REDUND_UNREPLICABLE} BOOL;
		Di_P_gas_low : {REDUND_UNREPLICABLE} BOOL;
		Di_P_gas_high : {REDUND_UNREPLICABLE} BOOL;
		Start : {REDUND_UNREPLICABLE} BOOL;
		Stop : {REDUND_UNREPLICABLE} BOOL;
	END_VAR
	VAR_OUTPUT
		Do_Spark : BOOL;
		Do_Valve : BOOL;
		Do_Lamp_P_Zapal_low : BOOL;
		Do_Lamp_FireON : BOOL;
		Do_Lamp_Alarm : BOOL;
	END_VAR
	VAR RETAIN
		Time_vent : USINT := 30;
		Time_firing : USINT := 90;
		Time_stabiliz : USINT := 30;
		Time_spark_off : USINT := 10;
		Time_spark_on : USINT := 15;
		Time_after_alarm : USINT := 90;
	END_VAR
	VAR
		Warning_1 : BOOL;
		Warning_2 : BOOL;
		step : USINT;
		Alarm : USINT;
		firing_count : USINT;
		Timer_vent : TON := (IN:=FALSE);
		Timer_firing : TON := (IN:=FALSE);
		Timer_stabiliz : TON := (IN:=FALSE);
		Timer_spark_off : TON := (IN:=FALSE);
		Timer_spark_on : TON := (IN:=FALSE);
		Timer_after_alarm : TON := (IN:=FALSE);
	END_VAR
END_FUNCTION_BLOCK

{REDUND_OK} FUNCTION_BLOCK FSwitch (*Switch*) (*$GROUP=User,$CAT=User,$GROUPICON=User.png,$CATICON=User.png*)
	VAR_INPUT
		Start_1 : BOOL;
		Start_2 : BOOL;
		Stop : BOOL;
		RunDI_1 : BOOL;
		RunDI_2 : BOOL;
		Reset : BOOL;
	END_VAR
	VAR_INPUT RETAIN
		Block_1 : BOOL;
		Block_2 : BOOL;
		Block_Stop : BOOL;
		Block : BOOL;
		Imitation : BOOL; (*Имитация*)
	END_VAR
	VAR_INPUT
		ResetMH : BOOL;
	END_VAR
	VAR_OUTPUT
		StartDO_1 : BOOL;
		StartDO_2 : BOOL;
		StopDO : BOOL;
		Status : UINT;
		Started_1 : BOOL;
		Started_2 : BOOL;
		Stopped : BOOL;
	END_VAR
	VAR RETAIN
		Timeout : BOOL;
	END_VAR
	VAR
		T : TON;
		Starting_2 : BOOL;
		Starting_1 : BOOL;
	END_VAR
END_FUNCTION_BLOCK

{REDUND_OK} FUNCTION_BLOCK fCmdCOM (*MBRTU Comand to opened interface*) (*$GROUP=User,$CAT=User,$GROUPICON=User.png,$CATICON=User.png*)
	VAR_INPUT
		ident : UDINT;
		pData : UDINT;
		offset : UINT;
		node : USINT;
		cmd : USINT;
		length : USINT;
	END_VAR
	VAR_OUTPUT
		status : UINT;
	END_VAR
	VAR
		MBMCmd_0 : MBMCmd;
	END_VAR
END_FUNCTION_BLOCK

{REDUND_OK} FUNCTION_BLOCK fOpenCOM (*Opens physical communication interface *) (*$GROUP=User,$CAT=User,$GROUPICON=User.png,$CATICON=User.png*)
	VAR_INPUT RETAIN
		enable : BOOL;
		Device : UDINT;
		Mode : UDINT;
		Config : UDINT;
	END_VAR
	VAR_OUTPUT
		status : UINT;
		ident : UDINT;
	END_VAR
	VAR
		MBMOpen_0 : MBMOpen;
	END_VAR
END_FUNCTION_BLOCK

{REDUND_OK} FUNCTION_BLOCK fCloseCOM (*Closes opened communication interface*) (*$GROUP=User,$CAT=User,$GROUPICON=User.png,$CATICON=User.png*)
	VAR_INPUT
		enable : BOOL;
		ident : UDINT;
	END_VAR
	VAR_OUTPUT
		status : UINT;
	END_VAR
	VAR
		MBMClose_0 : MBMClose;
	END_VAR
END_FUNCTION_BLOCK

{REDUND_OK} FUNCTION_BLOCK FAlarm (*Alarm with delay*) (*$GROUP=User,$CAT=User,$GROUPICON=User.png,$CATICON=User.png*)
	VAR_INPUT
		IN : UINT; (*Входное слово(побитово можно завести 15 аварий,1 бит на 1 аварию)*)
		EN : UINT; (*Слово управления(каждый бит включает/отключает отработку аварии бита входного слова)*)
		Ack : BOOL; (*Квитирование*)
		Delay : UINT; (*Время задержки*)
	END_VAR
	VAR_OUTPUT
		OUT_int : UINT; (*Результат побитово (1-ПАЗ сработал,0-ПАЗ не сработал)*)
		OUT : BOOL; (*Результат(1-ПАЗ сработал,0-ПАЗ не сработал)*)
		Result : UINT;
	END_VAR
	VAR RETAIN
		Timer : TON;
	END_VAR
END_FUNCTION_BLOCK

{REDUND_OK} FUNCTION_BLOCK UVP_RTU (*UVP over RTU*) (*$GROUP=User,$CAT=User,$GROUPICON=User.png,$CATICON=User.png*)
	VAR_INPUT
		pPort : UDINT;
	END_VAR
	VAR
		status : UINT;
		state : UINT;
		step : USINT;
		req_3x : mbReadHoldingRegs;
		req_4x : mbReadInputRegs;
		req_6x : mbWriteSingleReg;
		req_16x : mbWriteMultipleRegs;
		UVP_Data : tUVP_Data := (NTP:=(cmd:=13579,IpAddress1:=192,IpAddress2:=168,IpAddress3:=50,IpAddress4:=12));
		curTP : USINT;
		Timeout_T : TON;
	END_VAR
END_FUNCTION_BLOCK

{REDUND_OK} FUNCTION_BLOCK mbReadHoldingRegs (* *) (*$GROUP=User,$CAT=User,$GROUPICON=User.png,$CATICON=User.png*)
	VAR_INPUT
		enable : BOOL;
		pStation : UDINT;
		pData : UDINT;
		startAddress : UINT;
		nrRegisters : USINT;
		dataSize : USINT;
	END_VAR
	VAR_OUTPUT
		status : UINT;
	END_VAR
	VAR
		CmdCOM : fCmdCOM;
	END_VAR
END_FUNCTION_BLOCK

{REDUND_OK} FUNCTION_BLOCK mbReadInputRegs (* *) (*$GROUP=User,$CAT=User,$GROUPICON=User.png,$CATICON=User.png*)
	VAR_INPUT
		enable : BOOL;
		pStation : UDINT;
		pData : UDINT;
		startAddress : UINT;
		nrRegisters : USINT;
		dataSize : USINT;
	END_VAR
	VAR_OUTPUT
		status : UINT;
	END_VAR
	VAR
		CmdCOM : fCmdCOM;
	END_VAR
END_FUNCTION_BLOCK

{REDUND_OK} FUNCTION_BLOCK mbWriteSingleReg (* *) (*$GROUP=User,$CAT=User,$GROUPICON=User.png,$CATICON=User.png*)
	VAR_INPUT
		enable : BOOL;
		pStation : UDINT;
		pData : UDINT;
		startAddress : UINT;
		nrRegisters : USINT;
		dataSize : USINT;
	END_VAR
	VAR_OUTPUT
		status : UINT;
	END_VAR
	VAR
		CmdCOM : fCmdCOM;
	END_VAR
END_FUNCTION_BLOCK

{REDUND_OK} FUNCTION_BLOCK mbWriteMultipleRegs (* *) (*$GROUP=User,$CAT=User,$GROUPICON=User.png,$CATICON=User.png*)
	VAR_INPUT
		enable : BOOL;
		pStation : UDINT;
		pData : UDINT;
		startAddress : UINT;
		nrRegisters : USINT;
		dataSize : USINT;
	END_VAR
	VAR_OUTPUT
		status : UINT;
	END_VAR
	VAR
		CmdCOM : fCmdCOM;
	END_VAR
END_FUNCTION_BLOCK

{REDUND_OK} FUNCTION_BLOCK ATV_Control (*Управление ПЧ через Модбас*) (*$GROUP=User,$CAT=User,$GROUPICON=User.png,$CATICON=User.png*)
	VAR_INPUT
		PortIdent : UDINT;
		MB_Addr : USINT;
		cmdStart : BOOL;
		cmdStop : BOOL;
		cmdResetAlarm : BOOL;
		cmdQckStop : BOOL;
		IN_Freq : REAL;
	END_VAR
	VAR_OUTPUT
		stStarted : BOOL;
		stStopped : BOOL;
		stAlarm : BOOL;
		OUT_Freq : REAL;
	END_VAR
	VAR
		CmdCOM : MBMCmd;
		CMD : UINT;
		HMIS : UINT;
		LFR : UINT;
		RFR : UINT;
		step : USINT;
		step_old : USINT;
	END_VAR
END_FUNCTION_BLOCK

{REDUND_OK} FUNCTION_BLOCK fAuma_MB (*AUMA через Модбас*) (*$GROUP=User,$CAT=User,$GROUPICON=User.png,$CATICON=User.png*)
	VAR_INPUT
		mode : USINT;
		mbAddr : USINT;
		cmd : UINT; (*бит0-Открыть, бит1- Закрыть, бит3-Сброс*)
		setPosition : REAL;
		identCOM : UDINT;
	END_VAR
	VAR_OUTPUT
		state : UINT;
		curPosition : REAL; (*бит0-Открыт,бит1-Закрыт,бит3-Местный,бит4-Открывается,бит5-Закрывается*)
	END_VAR
	VAR
		step : USINT;
		cmd_old : UINT;
		CmdCOM : fCmdCOM;
		read : tAuma_read;
		write : tAuma_write;
	END_VAR
END_FUNCTION_BLOCK
```

- FPostGassing.st (not readable text: treated as protected, skipped)
